eRFID[68].nCardNumber;eRFID[68].bCapCorrectChecked;	eRFID[68].bCapCorrectCheckCameraOK;		eRFID[68].bCapCorrectCheckCameraChecked;		eRFID[68].bCapCorrectCapOn;eRFID[68].bCapCorrectNOK; eRFID[68].bFormPresent; eRFID[68].bBottlePresent; eRFID[68].bDosingTwoPhases; eRFID[68].nDispencerNr; eRFID[68].nDispencerNrSecondPhase; eRFID[68].lrDoseVolumeSV; eRFID[68].lrDoseVolumeCV; eRFID[68].lrDoseVolumeSVSecondPhase; eRFID[68].lrDoseVolumeCVSecondPhase; eRFID[68].bDosed;	eRFID[68].bDoseAborted; eRFID[68].bWeighed; eRFID[68].lrWeightSV; eRFID[68].lrWeightCV; eRFID[68].lrWeightMeasuredCV; eRFID[68].bWeightOK; eRFID[68].bCapPutted; eRFID[68].bCapChecked; eRFID[68].bCapOK; eRFID[68].bCapGripperScrewed; eRFID[68].bCapGripperScrewAborted; eRFID[68].bBottleTransferedToExit; eRFID[68].bBottleTransferedToLabeler; eRFID[68].lrWeightDif; eRFID[68].lrMinWeightCV;eRFID[68].lrMaxWeightCV;
eRFID[69].nCardNumber;eRFID[69].bCapCorrectChecked;	eRFID[69].bCapCorrectCheckCameraOK;		eRFID[69].bCapCorrectCheckCameraChecked;		eRFID[69].bCapCorrectCapOn;eRFID[69].bCapCorrectNOK; eRFID[69].bFormPresent; eRFID[69].bBottlePresent; eRFID[69].bDosingTwoPhases; eRFID[69].nDispencerNr; eRFID[69].nDispencerNrSecondPhase; eRFID[69].lrDoseVolumeSV; eRFID[69].lrDoseVolumeCV; eRFID[69].lrDoseVolumeSVSecondPhase; eRFID[69].lrDoseVolumeCVSecondPhase; eRFID[69].bDosed;	eRFID[69].bDoseAborted; eRFID[69].bWeighed; eRFID[69].lrWeightSV; eRFID[69].lrWeightCV; eRFID[69].lrWeightMeasuredCV; eRFID[69].bWeightOK; eRFID[69].bCapPutted; eRFID[69].bCapChecked; eRFID[69].bCapOK; eRFID[69].bCapGripperScrewed; eRFID[69].bCapGripperScrewAborted; eRFID[69].bBottleTransferedToExit; eRFID[69].bBottleTransferedToLabeler; eRFID[69].lrWeightDif; eRFID[69].lrMinWeightCV;eRFID[69].lrMaxWeightCV;
eRFID[70].nCardNumber;eRFID[70].bCapCorrectChecked;	eRFID[70].bCapCorrectCheckCameraOK;		eRFID[70].bCapCorrectCheckCameraChecked;		eRFID[70].bCapCorrectCapOn;eRFID[70].bCapCorrectNOK; eRFID[70].bFormPresent; eRFID[70].bBottlePresent; eRFID[70].bDosingTwoPhases; eRFID[70].nDispencerNr; eRFID[70].nDispencerNrSecondPhase; eRFID[70].lrDoseVolumeSV; eRFID[70].lrDoseVolumeCV; eRFID[70].lrDoseVolumeSVSecondPhase; eRFID[70].lrDoseVolumeCVSecondPhase; eRFID[70].bDosed;	eRFID[70].bDoseAborted; eRFID[70].bWeighed; eRFID[70].lrWeightSV; eRFID[70].lrWeightCV; eRFID[70].lrWeightMeasuredCV; eRFID[70].bWeightOK; eRFID[70].bCapPutted; eRFID[70].bCapChecked; eRFID[70].bCapOK; eRFID[70].bCapGripperScrewed; eRFID[70].bCapGripperScrewAborted; eRFID[70].bBottleTransferedToExit; eRFID[70].bBottleTransferedToLabeler; eRFID[70].lrWeightDif; eRFID[70].lrMinWeightCV;eRFID[70].lrMaxWeightCV;
eRFID[71].nCardNumber;eRFID[71].bCapCorrectChecked;	eRFID[71].bCapCorrectCheckCameraOK;		eRFID[71].bCapCorrectCheckCameraChecked;		eRFID[71].bCapCorrectCapOn;eRFID[71].bCapCorrectNOK; eRFID[71].bFormPresent; eRFID[71].bBottlePresent; eRFID[71].bDosingTwoPhases; eRFID[71].nDispencerNr; eRFID[71].nDispencerNrSecondPhase; eRFID[71].lrDoseVolumeSV; eRFID[71].lrDoseVolumeCV; eRFID[71].lrDoseVolumeSVSecondPhase; eRFID[71].lrDoseVolumeCVSecondPhase; eRFID[71].bDosed;	eRFID[71].bDoseAborted; eRFID[71].bWeighed; eRFID[71].lrWeightSV; eRFID[71].lrWeightCV; eRFID[71].lrWeightMeasuredCV; eRFID[71].bWeightOK; eRFID[71].bCapPutted; eRFID[71].bCapChecked; eRFID[71].bCapOK; eRFID[71].bCapGripperScrewed; eRFID[71].bCapGripperScrewAborted; eRFID[71].bBottleTransferedToExit; eRFID[71].bBottleTransferedToLabeler; eRFID[71].lrWeightDif; eRFID[71].lrMinWeightCV;eRFID[71].lrMaxWeightCV;
eRFID[72].nCardNumber;eRFID[72].bCapCorrectChecked;	eRFID[72].bCapCorrectCheckCameraOK;		eRFID[72].bCapCorrectCheckCameraChecked;		eRFID[72].bCapCorrectCapOn;eRFID[72].bCapCorrectNOK; eRFID[72].bFormPresent; eRFID[72].bBottlePresent; eRFID[72].bDosingTwoPhases; eRFID[72].nDispencerNr; eRFID[72].nDispencerNrSecondPhase; eRFID[72].lrDoseVolumeSV; eRFID[72].lrDoseVolumeCV; eRFID[72].lrDoseVolumeSVSecondPhase; eRFID[72].lrDoseVolumeCVSecondPhase; eRFID[72].bDosed;	eRFID[72].bDoseAborted; eRFID[72].bWeighed; eRFID[72].lrWeightSV; eRFID[72].lrWeightCV; eRFID[72].lrWeightMeasuredCV; eRFID[72].bWeightOK; eRFID[72].bCapPutted; eRFID[72].bCapChecked; eRFID[72].bCapOK; eRFID[72].bCapGripperScrewed; eRFID[72].bCapGripperScrewAborted; eRFID[72].bBottleTransferedToExit; eRFID[72].bBottleTransferedToLabeler; eRFID[72].lrWeightDif; eRFID[72].lrMinWeightCV;eRFID[72].lrMaxWeightCV;
eRFID[73].nCardNumber;eRFID[73].bCapCorrectChecked;	eRFID[73].bCapCorrectCheckCameraOK;		eRFID[73].bCapCorrectCheckCameraChecked;		eRFID[73].bCapCorrectCapOn;eRFID[73].bCapCorrectNOK; eRFID[73].bFormPresent; eRFID[73].bBottlePresent; eRFID[73].bDosingTwoPhases; eRFID[73].nDispencerNr; eRFID[73].nDispencerNrSecondPhase; eRFID[73].lrDoseVolumeSV; eRFID[73].lrDoseVolumeCV; eRFID[73].lrDoseVolumeSVSecondPhase; eRFID[73].lrDoseVolumeCVSecondPhase; eRFID[73].bDosed;	eRFID[73].bDoseAborted; eRFID[73].bWeighed; eRFID[73].lrWeightSV; eRFID[73].lrWeightCV; eRFID[73].lrWeightMeasuredCV; eRFID[73].bWeightOK; eRFID[73].bCapPutted; eRFID[73].bCapChecked; eRFID[73].bCapOK; eRFID[73].bCapGripperScrewed; eRFID[73].bCapGripperScrewAborted; eRFID[73].bBottleTransferedToExit; eRFID[73].bBottleTransferedToLabeler; eRFID[73].lrWeightDif; eRFID[73].lrMinWeightCV;eRFID[73].lrMaxWeightCV;
eRFID[74].nCardNumber;eRFID[74].bCapCorrectChecked;	eRFID[74].bCapCorrectCheckCameraOK;		eRFID[74].bCapCorrectCheckCameraChecked;		eRFID[74].bCapCorrectCapOn;eRFID[74].bCapCorrectNOK; eRFID[74].bFormPresent; eRFID[74].bBottlePresent; eRFID[74].bDosingTwoPhases; eRFID[74].nDispencerNr; eRFID[74].nDispencerNrSecondPhase; eRFID[74].lrDoseVolumeSV; eRFID[74].lrDoseVolumeCV; eRFID[74].lrDoseVolumeSVSecondPhase; eRFID[74].lrDoseVolumeCVSecondPhase; eRFID[74].bDosed;	eRFID[74].bDoseAborted; eRFID[74].bWeighed; eRFID[74].lrWeightSV; eRFID[74].lrWeightCV; eRFID[74].lrWeightMeasuredCV; eRFID[74].bWeightOK; eRFID[74].bCapPutted; eRFID[74].bCapChecked; eRFID[74].bCapOK; eRFID[74].bCapGripperScrewed; eRFID[74].bCapGripperScrewAborted; eRFID[74].bBottleTransferedToExit; eRFID[74].bBottleTransferedToLabeler; eRFID[74].lrWeightDif; eRFID[74].lrMinWeightCV;eRFID[74].lrMaxWeightCV;
eRFID[75].nCardNumber;eRFID[75].bCapCorrectChecked;	eRFID[75].bCapCorrectCheckCameraOK;		eRFID[75].bCapCorrectCheckCameraChecked;		eRFID[75].bCapCorrectCapOn;eRFID[75].bCapCorrectNOK; eRFID[75].bFormPresent; eRFID[75].bBottlePresent; eRFID[75].bDosingTwoPhases; eRFID[75].nDispencerNr; eRFID[75].nDispencerNrSecondPhase; eRFID[75].lrDoseVolumeSV; eRFID[75].lrDoseVolumeCV; eRFID[75].lrDoseVolumeSVSecondPhase; eRFID[75].lrDoseVolumeCVSecondPhase; eRFID[75].bDosed;	eRFID[75].bDoseAborted; eRFID[75].bWeighed; eRFID[75].lrWeightSV; eRFID[75].lrWeightCV; eRFID[75].lrWeightMeasuredCV; eRFID[75].bWeightOK; eRFID[75].bCapPutted; eRFID[75].bCapChecked; eRFID[75].bCapOK; eRFID[75].bCapGripperScrewed; eRFID[75].bCapGripperScrewAborted; eRFID[75].bBottleTransferedToExit; eRFID[75].bBottleTransferedToLabeler; eRFID[75].lrWeightDif; eRFID[75].lrMinWeightCV;eRFID[75].lrMaxWeightCV;
eRFID[76].nCardNumber;eRFID[76].bCapCorrectChecked;	eRFID[76].bCapCorrectCheckCameraOK;		eRFID[76].bCapCorrectCheckCameraChecked;		eRFID[76].bCapCorrectCapOn;eRFID[76].bCapCorrectNOK; eRFID[76].bFormPresent; eRFID[76].bBottlePresent; eRFID[76].bDosingTwoPhases; eRFID[76].nDispencerNr; eRFID[76].nDispencerNrSecondPhase; eRFID[76].lrDoseVolumeSV; eRFID[76].lrDoseVolumeCV; eRFID[76].lrDoseVolumeSVSecondPhase; eRFID[76].lrDoseVolumeCVSecondPhase; eRFID[76].bDosed;	eRFID[76].bDoseAborted; eRFID[76].bWeighed; eRFID[76].lrWeightSV; eRFID[76].lrWeightCV; eRFID[76].lrWeightMeasuredCV; eRFID[76].bWeightOK; eRFID[76].bCapPutted; eRFID[76].bCapChecked; eRFID[76].bCapOK; eRFID[76].bCapGripperScrewed; eRFID[76].bCapGripperScrewAborted; eRFID[76].bBottleTransferedToExit; eRFID[76].bBottleTransferedToLabeler; eRFID[76].lrWeightDif; eRFID[76].lrMinWeightCV;eRFID[76].lrMaxWeightCV;
eRFID[77].nCardNumber;eRFID[77].bCapCorrectChecked;	eRFID[77].bCapCorrectCheckCameraOK;		eRFID[77].bCapCorrectCheckCameraChecked;		eRFID[77].bCapCorrectCapOn;eRFID[77].bCapCorrectNOK; eRFID[77].bFormPresent; eRFID[77].bBottlePresent; eRFID[77].bDosingTwoPhases; eRFID[77].nDispencerNr; eRFID[77].nDispencerNrSecondPhase; eRFID[77].lrDoseVolumeSV; eRFID[77].lrDoseVolumeCV; eRFID[77].lrDoseVolumeSVSecondPhase; eRFID[77].lrDoseVolumeCVSecondPhase; eRFID[77].bDosed;	eRFID[77].bDoseAborted; eRFID[77].bWeighed; eRFID[77].lrWeightSV; eRFID[77].lrWeightCV; eRFID[77].lrWeightMeasuredCV; eRFID[77].bWeightOK; eRFID[77].bCapPutted; eRFID[77].bCapChecked; eRFID[77].bCapOK; eRFID[77].bCapGripperScrewed; eRFID[77].bCapGripperScrewAborted; eRFID[77].bBottleTransferedToExit; eRFID[77].bBottleTransferedToLabeler; eRFID[77].lrWeightDif; eRFID[77].lrMinWeightCV;eRFID[77].lrMaxWeightCV;
eRFID[78].nCardNumber;eRFID[78].bCapCorrectChecked;	eRFID[78].bCapCorrectCheckCameraOK;		eRFID[78].bCapCorrectCheckCameraChecked;		eRFID[78].bCapCorrectCapOn;eRFID[78].bCapCorrectNOK; eRFID[78].bFormPresent; eRFID[78].bBottlePresent; eRFID[78].bDosingTwoPhases; eRFID[78].nDispencerNr; eRFID[78].nDispencerNrSecondPhase; eRFID[78].lrDoseVolumeSV; eRFID[78].lrDoseVolumeCV; eRFID[78].lrDoseVolumeSVSecondPhase; eRFID[78].lrDoseVolumeCVSecondPhase; eRFID[78].bDosed;	eRFID[78].bDoseAborted; eRFID[78].bWeighed; eRFID[78].lrWeightSV; eRFID[78].lrWeightCV; eRFID[78].lrWeightMeasuredCV; eRFID[78].bWeightOK; eRFID[78].bCapPutted; eRFID[78].bCapChecked; eRFID[78].bCapOK; eRFID[78].bCapGripperScrewed; eRFID[78].bCapGripperScrewAborted; eRFID[78].bBottleTransferedToExit; eRFID[78].bBottleTransferedToLabeler; eRFID[78].lrWeightDif; eRFID[78].lrMinWeightCV;eRFID[78].lrMaxWeightCV;
eRFID[79].nCardNumber;eRFID[79].bCapCorrectChecked;	eRFID[79].bCapCorrectCheckCameraOK;		eRFID[79].bCapCorrectCheckCameraChecked;		eRFID[79].bCapCorrectCapOn;eRFID[79].bCapCorrectNOK; eRFID[79].bFormPresent; eRFID[79].bBottlePresent; eRFID[79].bDosingTwoPhases; eRFID[79].nDispencerNr; eRFID[79].nDispencerNrSecondPhase; eRFID[79].lrDoseVolumeSV; eRFID[79].lrDoseVolumeCV; eRFID[79].lrDoseVolumeSVSecondPhase; eRFID[79].lrDoseVolumeCVSecondPhase; eRFID[79].bDosed;	eRFID[79].bDoseAborted; eRFID[79].bWeighed; eRFID[79].lrWeightSV; eRFID[79].lrWeightCV; eRFID[79].lrWeightMeasuredCV; eRFID[79].bWeightOK; eRFID[79].bCapPutted; eRFID[79].bCapChecked; eRFID[79].bCapOK; eRFID[79].bCapGripperScrewed; eRFID[79].bCapGripperScrewAborted; eRFID[79].bBottleTransferedToExit; eRFID[79].bBottleTransferedToLabeler; eRFID[79].lrWeightDif; eRFID[79].lrMinWeightCV;eRFID[79].lrMaxWeightCV;
eRFID[80].nCardNumber;eRFID[80].bCapCorrectChecked;	eRFID[80].bCapCorrectCheckCameraOK;		eRFID[80].bCapCorrectCheckCameraChecked;		eRFID[80].bCapCorrectCapOn;eRFID[80].bCapCorrectNOK; eRFID[80].bFormPresent; eRFID[80].bBottlePresent; eRFID[80].bDosingTwoPhases; eRFID[80].nDispencerNr; eRFID[80].nDispencerNrSecondPhase; eRFID[80].lrDoseVolumeSV; eRFID[80].lrDoseVolumeCV; eRFID[80].lrDoseVolumeSVSecondPhase; eRFID[80].lrDoseVolumeCVSecondPhase; eRFID[80].bDosed;	eRFID[80].bDoseAborted; eRFID[80].bWeighed; eRFID[80].lrWeightSV; eRFID[80].lrWeightCV; eRFID[80].lrWeightMeasuredCV; eRFID[80].bWeightOK; eRFID[80].bCapPutted; eRFID[80].bCapChecked; eRFID[80].bCapOK; eRFID[80].bCapGripperScrewed; eRFID[80].bCapGripperScrewAborted; eRFID[80].bBottleTransferedToExit; eRFID[80].bBottleTransferedToLabeler; eRFID[80].lrWeightDif; eRFID[80].lrMinWeightCV;eRFID[80].lrMaxWeightCV;
eRFID[81].nCardNumber;eRFID[81].bCapCorrectChecked;	eRFID[81].bCapCorrectCheckCameraOK;		eRFID[81].bCapCorrectCheckCameraChecked;		eRFID[81].bCapCorrectCapOn;eRFID[81].bCapCorrectNOK; eRFID[81].bFormPresent; eRFID[81].bBottlePresent; eRFID[81].bDosingTwoPhases; eRFID[81].nDispencerNr; eRFID[81].nDispencerNrSecondPhase; eRFID[81].lrDoseVolumeSV; eRFID[81].lrDoseVolumeCV; eRFID[81].lrDoseVolumeSVSecondPhase; eRFID[81].lrDoseVolumeCVSecondPhase; eRFID[81].bDosed;	eRFID[81].bDoseAborted; eRFID[81].bWeighed; eRFID[81].lrWeightSV; eRFID[81].lrWeightCV; eRFID[81].lrWeightMeasuredCV; eRFID[81].bWeightOK; eRFID[81].bCapPutted; eRFID[81].bCapChecked; eRFID[81].bCapOK; eRFID[81].bCapGripperScrewed; eRFID[81].bCapGripperScrewAborted; eRFID[81].bBottleTransferedToExit; eRFID[81].bBottleTransferedToLabeler; eRFID[81].lrWeightDif; eRFID[81].lrMinWeightCV;eRFID[81].lrMaxWeightCV;
eRFID[82].nCardNumber;eRFID[82].bCapCorrectChecked;	eRFID[82].bCapCorrectCheckCameraOK;		eRFID[82].bCapCorrectCheckCameraChecked;		eRFID[82].bCapCorrectCapOn;eRFID[82].bCapCorrectNOK; eRFID[82].bFormPresent; eRFID[82].bBottlePresent; eRFID[82].bDosingTwoPhases; eRFID[82].nDispencerNr; eRFID[82].nDispencerNrSecondPhase; eRFID[82].lrDoseVolumeSV; eRFID[82].lrDoseVolumeCV; eRFID[82].lrDoseVolumeSVSecondPhase; eRFID[82].lrDoseVolumeCVSecondPhase; eRFID[82].bDosed;	eRFID[82].bDoseAborted; eRFID[82].bWeighed; eRFID[82].lrWeightSV; eRFID[82].lrWeightCV; eRFID[82].lrWeightMeasuredCV; eRFID[82].bWeightOK; eRFID[82].bCapPutted; eRFID[82].bCapChecked; eRFID[82].bCapOK; eRFID[82].bCapGripperScrewed; eRFID[82].bCapGripperScrewAborted; eRFID[82].bBottleTransferedToExit; eRFID[82].bBottleTransferedToLabeler; eRFID[82].lrWeightDif; eRFID[82].lrMinWeightCV;eRFID[82].lrMaxWeightCV;
eRFID[83].nCardNumber;eRFID[83].bCapCorrectChecked;	eRFID[83].bCapCorrectCheckCameraOK;		eRFID[83].bCapCorrectCheckCameraChecked;		eRFID[83].bCapCorrectCapOn;eRFID[83].bCapCorrectNOK; eRFID[83].bFormPresent; eRFID[83].bBottlePresent; eRFID[83].bDosingTwoPhases; eRFID[83].nDispencerNr; eRFID[83].nDispencerNrSecondPhase; eRFID[83].lrDoseVolumeSV; eRFID[83].lrDoseVolumeCV; eRFID[83].lrDoseVolumeSVSecondPhase; eRFID[83].lrDoseVolumeCVSecondPhase; eRFID[83].bDosed;	eRFID[83].bDoseAborted; eRFID[83].bWeighed; eRFID[83].lrWeightSV; eRFID[83].lrWeightCV; eRFID[83].lrWeightMeasuredCV; eRFID[83].bWeightOK; eRFID[83].bCapPutted; eRFID[83].bCapChecked; eRFID[83].bCapOK; eRFID[83].bCapGripperScrewed; eRFID[83].bCapGripperScrewAborted; eRFID[83].bBottleTransferedToExit; eRFID[83].bBottleTransferedToLabeler; eRFID[83].lrWeightDif; eRFID[83].lrMinWeightCV;eRFID[83].lrMaxWeightCV;
eRFID[84].nCardNumber;eRFID[84].bCapCorrectChecked;	eRFID[84].bCapCorrectCheckCameraOK;		eRFID[84].bCapCorrectCheckCameraChecked;		eRFID[84].bCapCorrectCapOn;eRFID[84].bCapCorrectNOK; eRFID[84].bFormPresent; eRFID[84].bBottlePresent; eRFID[84].bDosingTwoPhases; eRFID[84].nDispencerNr; eRFID[84].nDispencerNrSecondPhase; eRFID[84].lrDoseVolumeSV; eRFID[84].lrDoseVolumeCV; eRFID[84].lrDoseVolumeSVSecondPhase; eRFID[84].lrDoseVolumeCVSecondPhase; eRFID[84].bDosed;	eRFID[84].bDoseAborted; eRFID[84].bWeighed; eRFID[84].lrWeightSV; eRFID[84].lrWeightCV; eRFID[84].lrWeightMeasuredCV; eRFID[84].bWeightOK; eRFID[84].bCapPutted; eRFID[84].bCapChecked; eRFID[84].bCapOK; eRFID[84].bCapGripperScrewed; eRFID[84].bCapGripperScrewAborted; eRFID[84].bBottleTransferedToExit; eRFID[84].bBottleTransferedToLabeler; eRFID[84].lrWeightDif; eRFID[84].lrMinWeightCV;eRFID[84].lrMaxWeightCV;
eRFID[85].nCardNumber;eRFID[85].bCapCorrectChecked;	eRFID[85].bCapCorrectCheckCameraOK;		eRFID[85].bCapCorrectCheckCameraChecked;		eRFID[85].bCapCorrectCapOn;eRFID[85].bCapCorrectNOK; eRFID[85].bFormPresent; eRFID[85].bBottlePresent; eRFID[85].bDosingTwoPhases; eRFID[85].nDispencerNr; eRFID[85].nDispencerNrSecondPhase; eRFID[85].lrDoseVolumeSV; eRFID[85].lrDoseVolumeCV; eRFID[85].lrDoseVolumeSVSecondPhase; eRFID[85].lrDoseVolumeCVSecondPhase; eRFID[85].bDosed;	eRFID[85].bDoseAborted; eRFID[85].bWeighed; eRFID[85].lrWeightSV; eRFID[85].lrWeightCV; eRFID[85].lrWeightMeasuredCV; eRFID[85].bWeightOK; eRFID[85].bCapPutted; eRFID[85].bCapChecked; eRFID[85].bCapOK; eRFID[85].bCapGripperScrewed; eRFID[85].bCapGripperScrewAborted; eRFID[85].bBottleTransferedToExit; eRFID[85].bBottleTransferedToLabeler; eRFID[85].lrWeightDif; eRFID[85].lrMinWeightCV;eRFID[85].lrMaxWeightCV;
eRFID[86].nCardNumber;eRFID[86].bCapCorrectChecked;	eRFID[86].bCapCorrectCheckCameraOK;		eRFID[86].bCapCorrectCheckCameraChecked;		eRFID[86].bCapCorrectCapOn;eRFID[86].bCapCorrectNOK; eRFID[86].bFormPresent; eRFID[86].bBottlePresent; eRFID[86].bDosingTwoPhases; eRFID[86].nDispencerNr; eRFID[86].nDispencerNrSecondPhase; eRFID[86].lrDoseVolumeSV; eRFID[86].lrDoseVolumeCV; eRFID[86].lrDoseVolumeSVSecondPhase; eRFID[86].lrDoseVolumeCVSecondPhase; eRFID[86].bDosed;	eRFID[86].bDoseAborted; eRFID[86].bWeighed; eRFID[86].lrWeightSV; eRFID[86].lrWeightCV; eRFID[86].lrWeightMeasuredCV; eRFID[86].bWeightOK; eRFID[86].bCapPutted; eRFID[86].bCapChecked; eRFID[86].bCapOK; eRFID[86].bCapGripperScrewed; eRFID[86].bCapGripperScrewAborted; eRFID[86].bBottleTransferedToExit; eRFID[86].bBottleTransferedToLabeler; eRFID[86].lrWeightDif; eRFID[86].lrMinWeightCV;eRFID[86].lrMaxWeightCV;
eRFID[87].nCardNumber;eRFID[87].bCapCorrectChecked;	eRFID[87].bCapCorrectCheckCameraOK;		eRFID[87].bCapCorrectCheckCameraChecked;		eRFID[87].bCapCorrectCapOn;eRFID[87].bCapCorrectNOK; eRFID[87].bFormPresent; eRFID[87].bBottlePresent; eRFID[87].bDosingTwoPhases; eRFID[87].nDispencerNr; eRFID[87].nDispencerNrSecondPhase; eRFID[87].lrDoseVolumeSV; eRFID[87].lrDoseVolumeCV; eRFID[87].lrDoseVolumeSVSecondPhase; eRFID[87].lrDoseVolumeCVSecondPhase; eRFID[87].bDosed;	eRFID[87].bDoseAborted; eRFID[87].bWeighed; eRFID[87].lrWeightSV; eRFID[87].lrWeightCV; eRFID[87].lrWeightMeasuredCV; eRFID[87].bWeightOK; eRFID[87].bCapPutted; eRFID[87].bCapChecked; eRFID[87].bCapOK; eRFID[87].bCapGripperScrewed; eRFID[87].bCapGripperScrewAborted; eRFID[87].bBottleTransferedToExit; eRFID[87].bBottleTransferedToLabeler; eRFID[87].lrWeightDif; eRFID[87].lrMinWeightCV;eRFID[87].lrMaxWeightCV;
eRFID[88].nCardNumber;eRFID[88].bCapCorrectChecked;	eRFID[88].bCapCorrectCheckCameraOK;		eRFID[88].bCapCorrectCheckCameraChecked;		eRFID[88].bCapCorrectCapOn;eRFID[88].bCapCorrectNOK; eRFID[88].bFormPresent; eRFID[88].bBottlePresent; eRFID[88].bDosingTwoPhases; eRFID[88].nDispencerNr; eRFID[88].nDispencerNrSecondPhase; eRFID[88].lrDoseVolumeSV; eRFID[88].lrDoseVolumeCV; eRFID[88].lrDoseVolumeSVSecondPhase; eRFID[88].lrDoseVolumeCVSecondPhase; eRFID[88].bDosed;	eRFID[88].bDoseAborted; eRFID[88].bWeighed; eRFID[88].lrWeightSV; eRFID[88].lrWeightCV; eRFID[88].lrWeightMeasuredCV; eRFID[88].bWeightOK; eRFID[88].bCapPutted; eRFID[88].bCapChecked; eRFID[88].bCapOK; eRFID[88].bCapGripperScrewed; eRFID[88].bCapGripperScrewAborted; eRFID[88].bBottleTransferedToExit; eRFID[88].bBottleTransferedToLabeler; eRFID[88].lrWeightDif; eRFID[88].lrMinWeightCV;eRFID[88].lrMaxWeightCV;
eRFID[89].nCardNumber;eRFID[89].bCapCorrectChecked;	eRFID[89].bCapCorrectCheckCameraOK;		eRFID[89].bCapCorrectCheckCameraChecked;		eRFID[89].bCapCorrectCapOn;eRFID[89].bCapCorrectNOK; eRFID[89].bFormPresent; eRFID[89].bBottlePresent; eRFID[89].bDosingTwoPhases; eRFID[89].nDispencerNr; eRFID[89].nDispencerNrSecondPhase; eRFID[89].lrDoseVolumeSV; eRFID[89].lrDoseVolumeCV; eRFID[89].lrDoseVolumeSVSecondPhase; eRFID[89].lrDoseVolumeCVSecondPhase; eRFID[89].bDosed;	eRFID[89].bDoseAborted; eRFID[89].bWeighed; eRFID[89].lrWeightSV; eRFID[89].lrWeightCV; eRFID[89].lrWeightMeasuredCV; eRFID[89].bWeightOK; eRFID[89].bCapPutted; eRFID[89].bCapChecked; eRFID[89].bCapOK; eRFID[89].bCapGripperScrewed; eRFID[89].bCapGripperScrewAborted; eRFID[89].bBottleTransferedToExit; eRFID[89].bBottleTransferedToLabeler; eRFID[89].lrWeightDif; eRFID[89].lrMinWeightCV;eRFID[89].lrMaxWeightCV;
eRFID[90].nCardNumber;eRFID[90].bCapCorrectChecked;	eRFID[90].bCapCorrectCheckCameraOK;		eRFID[90].bCapCorrectCheckCameraChecked;		eRFID[90].bCapCorrectCapOn;eRFID[90].bCapCorrectNOK; eRFID[90].bFormPresent; eRFID[90].bBottlePresent; eRFID[90].bDosingTwoPhases; eRFID[90].nDispencerNr; eRFID[90].nDispencerNrSecondPhase; eRFID[90].lrDoseVolumeSV; eRFID[90].lrDoseVolumeCV; eRFID[90].lrDoseVolumeSVSecondPhase; eRFID[90].lrDoseVolumeCVSecondPhase; eRFID[90].bDosed;	eRFID[90].bDoseAborted; eRFID[90].bWeighed; eRFID[90].lrWeightSV; eRFID[90].lrWeightCV; eRFID[90].lrWeightMeasuredCV; eRFID[90].bWeightOK; eRFID[90].bCapPutted; eRFID[90].bCapChecked; eRFID[90].bCapOK; eRFID[90].bCapGripperScrewed; eRFID[90].bCapGripperScrewAborted; eRFID[90].bBottleTransferedToExit; eRFID[90].bBottleTransferedToLabeler; eRFID[90].lrWeightDif; eRFID[90].lrMinWeightCV;eRFID[90].lrMaxWeightCV;
eRFID[91].nCardNumber;eRFID[91].bCapCorrectChecked;	eRFID[91].bCapCorrectCheckCameraOK;		eRFID[91].bCapCorrectCheckCameraChecked;		eRFID[91].bCapCorrectCapOn;eRFID[91].bCapCorrectNOK; eRFID[91].bFormPresent; eRFID[91].bBottlePresent; eRFID[91].bDosingTwoPhases; eRFID[91].nDispencerNr; eRFID[91].nDispencerNrSecondPhase; eRFID[91].lrDoseVolumeSV; eRFID[91].lrDoseVolumeCV; eRFID[91].lrDoseVolumeSVSecondPhase; eRFID[91].lrDoseVolumeCVSecondPhase; eRFID[91].bDosed;	eRFID[91].bDoseAborted; eRFID[91].bWeighed; eRFID[91].lrWeightSV; eRFID[91].lrWeightCV; eRFID[91].lrWeightMeasuredCV; eRFID[91].bWeightOK; eRFID[91].bCapPutted; eRFID[91].bCapChecked; eRFID[91].bCapOK; eRFID[91].bCapGripperScrewed; eRFID[91].bCapGripperScrewAborted; eRFID[91].bBottleTransferedToExit; eRFID[91].bBottleTransferedToLabeler; eRFID[91].lrWeightDif; eRFID[91].lrMinWeightCV;eRFID[91].lrMaxWeightCV;
eRFID[92].nCardNumber;eRFID[92].bCapCorrectChecked;	eRFID[92].bCapCorrectCheckCameraOK;		eRFID[92].bCapCorrectCheckCameraChecked;		eRFID[92].bCapCorrectCapOn;eRFID[92].bCapCorrectNOK; eRFID[92].bFormPresent; eRFID[92].bBottlePresent; eRFID[92].bDosingTwoPhases; eRFID[92].nDispencerNr; eRFID[92].nDispencerNrSecondPhase; eRFID[92].lrDoseVolumeSV; eRFID[92].lrDoseVolumeCV; eRFID[92].lrDoseVolumeSVSecondPhase; eRFID[92].lrDoseVolumeCVSecondPhase; eRFID[92].bDosed;	eRFID[92].bDoseAborted; eRFID[92].bWeighed; eRFID[92].lrWeightSV; eRFID[92].lrWeightCV; eRFID[92].lrWeightMeasuredCV; eRFID[92].bWeightOK; eRFID[92].bCapPutted; eRFID[92].bCapChecked; eRFID[92].bCapOK; eRFID[92].bCapGripperScrewed; eRFID[92].bCapGripperScrewAborted; eRFID[92].bBottleTransferedToExit; eRFID[92].bBottleTransferedToLabeler; eRFID[92].lrWeightDif; eRFID[92].lrMinWeightCV;eRFID[92].lrMaxWeightCV;
eRFID[93].nCardNumber;eRFID[93].bCapCorrectChecked;	eRFID[93].bCapCorrectCheckCameraOK;		eRFID[93].bCapCorrectCheckCameraChecked;		eRFID[93].bCapCorrectCapOn;eRFID[93].bCapCorrectNOK; eRFID[93].bFormPresent; eRFID[93].bBottlePresent; eRFID[93].bDosingTwoPhases; eRFID[93].nDispencerNr; eRFID[93].nDispencerNrSecondPhase; eRFID[93].lrDoseVolumeSV; eRFID[93].lrDoseVolumeCV; eRFID[93].lrDoseVolumeSVSecondPhase; eRFID[93].lrDoseVolumeCVSecondPhase; eRFID[93].bDosed;	eRFID[93].bDoseAborted; eRFID[93].bWeighed; eRFID[93].lrWeightSV; eRFID[93].lrWeightCV; eRFID[93].lrWeightMeasuredCV; eRFID[93].bWeightOK; eRFID[93].bCapPutted; eRFID[93].bCapChecked; eRFID[93].bCapOK; eRFID[93].bCapGripperScrewed; eRFID[93].bCapGripperScrewAborted; eRFID[93].bBottleTransferedToExit; eRFID[93].bBottleTransferedToLabeler; eRFID[93].lrWeightDif; eRFID[93].lrMinWeightCV;eRFID[93].lrMaxWeightCV;
eRFID[94].nCardNumber;eRFID[94].bCapCorrectChecked;	eRFID[94].bCapCorrectCheckCameraOK;		eRFID[94].bCapCorrectCheckCameraChecked;		eRFID[94].bCapCorrectCapOn;eRFID[94].bCapCorrectNOK; eRFID[94].bFormPresent; eRFID[94].bBottlePresent; eRFID[94].bDosingTwoPhases; eRFID[94].nDispencerNr; eRFID[94].nDispencerNrSecondPhase; eRFID[94].lrDoseVolumeSV; eRFID[94].lrDoseVolumeCV; eRFID[94].lrDoseVolumeSVSecondPhase; eRFID[94].lrDoseVolumeCVSecondPhase; eRFID[94].bDosed;	eRFID[94].bDoseAborted; eRFID[94].bWeighed; eRFID[94].lrWeightSV; eRFID[94].lrWeightCV; eRFID[94].lrWeightMeasuredCV; eRFID[94].bWeightOK; eRFID[94].bCapPutted; eRFID[94].bCapChecked; eRFID[94].bCapOK; eRFID[94].bCapGripperScrewed; eRFID[94].bCapGripperScrewAborted; eRFID[94].bBottleTransferedToExit; eRFID[94].bBottleTransferedToLabeler; eRFID[94].lrWeightDif; eRFID[94].lrMinWeightCV;eRFID[94].lrMaxWeightCV;
eRFID[95].nCardNumber;eRFID[95].bCapCorrectChecked;	eRFID[95].bCapCorrectCheckCameraOK;		eRFID[95].bCapCorrectCheckCameraChecked;		eRFID[95].bCapCorrectCapOn;eRFID[95].bCapCorrectNOK; eRFID[95].bFormPresent; eRFID[95].bBottlePresent; eRFID[95].bDosingTwoPhases; eRFID[95].nDispencerNr; eRFID[95].nDispencerNrSecondPhase; eRFID[95].lrDoseVolumeSV; eRFID[95].lrDoseVolumeCV; eRFID[95].lrDoseVolumeSVSecondPhase; eRFID[95].lrDoseVolumeCVSecondPhase; eRFID[95].bDosed;	eRFID[95].bDoseAborted; eRFID[95].bWeighed; eRFID[95].lrWeightSV; eRFID[95].lrWeightCV; eRFID[95].lrWeightMeasuredCV; eRFID[95].bWeightOK; eRFID[95].bCapPutted; eRFID[95].bCapChecked; eRFID[95].bCapOK; eRFID[95].bCapGripperScrewed; eRFID[95].bCapGripperScrewAborted; eRFID[95].bBottleTransferedToExit; eRFID[95].bBottleTransferedToLabeler; eRFID[95].lrWeightDif; eRFID[95].lrMinWeightCV;eRFID[95].lrMaxWeightCV;
eRFID[96].nCardNumber;eRFID[96].bCapCorrectChecked;	eRFID[96].bCapCorrectCheckCameraOK;		eRFID[96].bCapCorrectCheckCameraChecked;		eRFID[96].bCapCorrectCapOn;eRFID[96].bCapCorrectNOK; eRFID[96].bFormPresent; eRFID[96].bBottlePresent; eRFID[96].bDosingTwoPhases; eRFID[96].nDispencerNr; eRFID[96].nDispencerNrSecondPhase; eRFID[96].lrDoseVolumeSV; eRFID[96].lrDoseVolumeCV; eRFID[96].lrDoseVolumeSVSecondPhase; eRFID[96].lrDoseVolumeCVSecondPhase; eRFID[96].bDosed;	eRFID[96].bDoseAborted; eRFID[96].bWeighed; eRFID[96].lrWeightSV; eRFID[96].lrWeightCV; eRFID[96].lrWeightMeasuredCV; eRFID[96].bWeightOK; eRFID[96].bCapPutted; eRFID[96].bCapChecked; eRFID[96].bCapOK; eRFID[96].bCapGripperScrewed; eRFID[96].bCapGripperScrewAborted; eRFID[96].bBottleTransferedToExit; eRFID[96].bBottleTransferedToLabeler; eRFID[96].lrWeightDif; eRFID[96].lrMinWeightCV;eRFID[96].lrMaxWeightCV;
eRFID[97].nCardNumber;eRFID[97].bCapCorrectChecked;	eRFID[97].bCapCorrectCheckCameraOK;		eRFID[97].bCapCorrectCheckCameraChecked;		eRFID[97].bCapCorrectCapOn;eRFID[97].bCapCorrectNOK; eRFID[97].bFormPresent; eRFID[97].bBottlePresent; eRFID[97].bDosingTwoPhases; eRFID[97].nDispencerNr; eRFID[97].nDispencerNrSecondPhase; eRFID[97].lrDoseVolumeSV; eRFID[97].lrDoseVolumeCV; eRFID[97].lrDoseVolumeSVSecondPhase; eRFID[97].lrDoseVolumeCVSecondPhase; eRFID[97].bDosed;	eRFID[97].bDoseAborted; eRFID[97].bWeighed; eRFID[97].lrWeightSV; eRFID[97].lrWeightCV; eRFID[97].lrWeightMeasuredCV; eRFID[97].bWeightOK; eRFID[97].bCapPutted; eRFID[97].bCapChecked; eRFID[97].bCapOK; eRFID[97].bCapGripperScrewed; eRFID[97].bCapGripperScrewAborted; eRFID[97].bBottleTransferedToExit; eRFID[97].bBottleTransferedToLabeler; eRFID[97].lrWeightDif; eRFID[97].lrMinWeightCV;eRFID[97].lrMaxWeightCV;
eRFID[98].nCardNumber;eRFID[98].bCapCorrectChecked;	eRFID[98].bCapCorrectCheckCameraOK;		eRFID[98].bCapCorrectCheckCameraChecked;		eRFID[98].bCapCorrectCapOn;eRFID[98].bCapCorrectNOK; eRFID[98].bFormPresent; eRFID[98].bBottlePresent; eRFID[98].bDosingTwoPhases; eRFID[98].nDispencerNr; eRFID[98].nDispencerNrSecondPhase; eRFID[98].lrDoseVolumeSV; eRFID[98].lrDoseVolumeCV; eRFID[98].lrDoseVolumeSVSecondPhase; eRFID[98].lrDoseVolumeCVSecondPhase; eRFID[98].bDosed;	eRFID[98].bDoseAborted; eRFID[98].bWeighed; eRFID[98].lrWeightSV; eRFID[98].lrWeightCV; eRFID[98].lrWeightMeasuredCV; eRFID[98].bWeightOK; eRFID[98].bCapPutted; eRFID[98].bCapChecked; eRFID[98].bCapOK; eRFID[98].bCapGripperScrewed; eRFID[98].bCapGripperScrewAborted; eRFID[98].bBottleTransferedToExit; eRFID[98].bBottleTransferedToLabeler; eRFID[98].lrWeightDif; eRFID[98].lrMinWeightCV;eRFID[98].lrMaxWeightCV;
eRFID[99].nCardNumber;eRFID[99].bCapCorrectChecked;	eRFID[99].bCapCorrectCheckCameraOK;		eRFID[99].bCapCorrectCheckCameraChecked;		eRFID[99].bCapCorrectCapOn;eRFID[99].bCapCorrectNOK; eRFID[99].bFormPresent; eRFID[99].bBottlePresent; eRFID[99].bDosingTwoPhases; eRFID[99].nDispencerNr; eRFID[99].nDispencerNrSecondPhase; eRFID[99].lrDoseVolumeSV; eRFID[99].lrDoseVolumeCV; eRFID[99].lrDoseVolumeSVSecondPhase; eRFID[99].lrDoseVolumeCVSecondPhase; eRFID[99].bDosed;	eRFID[99].bDoseAborted; eRFID[99].bWeighed; eRFID[99].lrWeightSV; eRFID[99].lrWeightCV; eRFID[99].lrWeightMeasuredCV; eRFID[99].bWeightOK; eRFID[99].bCapPutted; eRFID[99].bCapChecked; eRFID[99].bCapOK; eRFID[99].bCapGripperScrewed; eRFID[99].bCapGripperScrewAborted; eRFID[99].bBottleTransferedToExit; eRFID[99].bBottleTransferedToLabeler; eRFID[99].lrWeightDif; eRFID[99].lrMinWeightCV;eRFID[99].lrMaxWeightCV;
eRFID[100].nCardNumber;eRFID[100].bCapCorrectChecked;eRFID[100].bCapCorrectCheckCameraOK;;	eRFID[100].bCapCorrectCheckCameraChecked;;		eRFID[100].bCapCorrectCapOn;eRFID[100].bCapCorrectNOK;eRFID[100].bFormPresent; eRFID[100].bBottlePresent; eRFID[100].bDosingTwoPhases; eRFID[100].nDispencerNr; eRFID[100].nDispencerNrSecondPhase; eRFID[100].lrDoseVolumeSV; eRFID[100].lrDoseVolumeCV; eRFID[100].lrDoseVolumeSVSecondPhase; eRFID[100].lrDoseVolumeCVSecondPhase; eRFID[100].bDoseAborted; eRFID[100].bWeighed; eRFID[100].lrWeightSV; eRFID[100].lrWeightCV; eRFID[100].lrWeightMeasuredCV; eRFID[100].bWeightOK; eRFID[100].bCapPutted; eRFID[100].bCapChecked; eRFID[100].bCapOK; eRFID[100].bCapGripperScrewed; eRFID[100].bCapGripperScrewAborted; eRFID[100].bBottleTransferedToExit; eRFID[100].bBottleTransferedToLabeler; eRFID[100].lrWeightDif; eRFID[100].lrMinWeightCV;eRFID[100].lrMinWeightCV;;


IF GVL.bV1Hz THEN
	FOR i := 1 TO 100 DO
		IF eRFID[i].nCardNumber = 544 THEN
			iPodglad := i;
		END_IF
	END_FOR
END_IF
IF iPodglad = 0 THEN
	 iPodglad := 100;
END_IF
;eRFID[iPodglad].nCardNumber;eRFID[iPodglad].bFormPresent;eRFID[iPodglad].bBottlePresent;eRFID[iPodglad].bWeighed;
;eRFID[iPodglad].bWeightOK;
;eRFID[iPodglad].bDosed;
;eRFID[iPodglad].bCapOK;
;eRFID[iPodglad].bCapCorrectCapOn;
;eRFID[iPodglad].bCapCorrectNOK;
;eRFID[iPodglad].bCapGripperScrewed;
;eRFID[iPodglad].bCapGripperScrewAborted;
;eRFID[iPodglad].bROPPPuttedChecked;
;eRFID[iPodglad].bROPPPutted;
;eRFID[iPodglad].bROPPCapped;
;eRFID[iPodglad].bROPPCappingAborted;
;eRFID[iPodglad].tROPPCappingTime;
;eRFID[iPodglad].bROPPCappingOK;
;eRFID[iPodglad].bROPPCappingChecked;
;eRFID[iPodglad].bCapSorterPutted;
;eRFID[iPodglad].bCapSorterPuttedAborted;
END_ACTION

ACTION aStatisticsROPP:

eUnderROPPPackageState[1].bROPPPuttedChecked;
eUnderROPPPackageState[1].bROPPPutted;
eUnderROPPPackageState[1].bROPPCapped;
eUnderROPPPackageState[1].bROPPCappingAborted;
eUnderROPPPackageState[1].tROPPCappingTime;
eUnderROPPPackageState[1].bROPPCappingOK;
eUnderROPPPackageState[1].bROPPCappingChecked;

eBeforeROPPCapControlPackageState[1].nID; eBeforeROPPCapControlPackageState[1].nCardNumber; eBeforeROPPCapControlPackageState[1].bFormPresent;eBeforeROPPCapControlPackageState[1].bBottlePresent;eBeforeROPPCapControlPackageState[1].bROPPPuttedChecked;	eBeforeROPPCapControlPackageState[1].bROPPPutted;

// [1..12] Strukura przed ROPP
eBeforeROPP2PackageState[3].nID; eBeforeROPP2PackageState[3].nCardNumber; eBeforeROPP2PackageState[3].bFormPresent; eBeforeROPP2PackageState[3].bBottlePresent;	eBeforeROPP2PackageState[3].bROPPPuttedChecked;	eBeforeROPP2PackageState[3].bROPPPutted;		 eBeforeROPP2PackageState[3].bDosingTwoPhases; eBeforeROPP2PackageState[3].lrDoseVolumeSV; eBeforeROPP2PackageState[3].lrDoseVolumeSVSecondPhase;  eBeforeROPP2PackageState[3].lrDoseVolumeCV; eBeforeROPP2PackageState[3].lrDoseVolumeCVSecondPhase; eBeforeROPP2PackageState[3].nDispencerNr; eBeforeROPP2PackageState[3].nDispencerNrSecondPhase; eBeforeROPP2PackageState[3].tDispencingTime; eBeforeROPP2PackageState[3].tDispencingTimeSecondPhase; eBeforeROPP2PackageState[3].bWeighed; eBeforeROPP2PackageState[2].bWeightOK; eBeforeROPP2PackageState[3].lrWeightSV; eBeforeROPP2PackageState[3].lrWeightMeasuredCV; eBeforeROPP2PackageState[3].lrWeightCV; eBeforeROPP2PackageState[3].bCapChecked;
eBeforeROPP2PackageState[2].nID; eBeforeROPP2PackageState[2].nCardNumber; eBeforeROPP2PackageState[2].bFormPresent; eBeforeROPP2PackageState[2].bBottlePresent;	eBeforeROPP2PackageState[2].bROPPPuttedChecked;	eBeforeROPP2PackageState[2].bROPPPutted;		 eBeforeROPP2PackageState[2].bDosingTwoPhases; eBeforeROPP2PackageState[2].lrDoseVolumeSV; eBeforeROPP2PackageState[2].lrDoseVolumeSVSecondPhase;  eBeforeROPP2PackageState[2].lrDoseVolumeCV; eBeforeROPP2PackageState[2].lrDoseVolumeCVSecondPhase; eBeforeROPP2PackageState[2].nDispencerNr; eBeforeROPP2PackageState[2].nDispencerNrSecondPhase; eBeforeROPP2PackageState[2].tDispencingTime; eBeforeROPP2PackageState[2].tDispencingTimeSecondPhase; eBeforeROPP2PackageState[2].bWeighed; eBeforeROPP2PackageState[2].bWeightOK; eBeforeROPP2PackageState[2].lrWeightSV; eBeforeROPP2PackageState[2].lrWeightMeasuredCV; eBeforeROPP2PackageState[2].lrWeightCV; eBeforeROPP2PackageState[2].bCapChecked;
eBeforeROPP2PackageState[1].nID; eBeforeROPP2PackageState[1].nCardNumber; eBeforeROPP2PackageState[1].bFormPresent; eBeforeROPP2PackageState[1].bBottlePresent;	eBeforeROPP2PackageState[1].bROPPPuttedChecked;	eBeforeROPP2PackageState[1].bROPPPutted;		 eBeforeROPP2PackageState[1].bDosingTwoPhases; eBeforeROPP2PackageState[1].lrDoseVolumeSV; eBeforeROPP2PackageState[1].lrDoseVolumeSVSecondPhase;  eBeforeROPP2PackageState[1].lrDoseVolumeCV; eBeforeROPP2PackageState[1].lrDoseVolumeCVSecondPhase; eBeforeROPP2PackageState[1].nDispencerNr; eBeforeROPP2PackageState[1].nDispencerNrSecondPhase; eBeforeROPP2PackageState[1].tDispencingTime; eBeforeROPP2PackageState[1].tDispencingTimeSecondPhase; eBeforeROPP2PackageState[1].bWeighed; eBeforeROPP2PackageState[1].bWeightOK; eBeforeROPP2PackageState[1].lrWeightSV; eBeforeROPP2PackageState[1].lrWeightMeasuredCV; eBeforeROPP2PackageState[1].lrWeightCV; eBeforeROPP2PackageState[1].bCapChecked;
eBeforeROPPPackageState[2].nID;  eBeforeROPPPackageState[2].nCardNumber;  eBeforeROPPPackageState[2].bFormPresent;  eBeforeROPPPackageState[2].bBottlePresent;	eBeforeROPPPackageState[2].bROPPPuttedChecked;	eBeforeROPPPackageState[2].bROPPPutted;		 eBeforeROPPPackageState[2].bDosingTwoPhases; eBeforeROPPPackageState[2].lrDoseVolumeSV; eBeforeROPPPackageState[2].lrDoseVolumeSVSecondPhase;  eBeforeROPPPackageState[2].lrDoseVolumeCV; eBeforeROPPPackageState[2].lrDoseVolumeCVSecondPhase; eBeforeROPPPackageState[2].nDispencerNr; eBeforeROPPPackageState[2].nDispencerNrSecondPhase; eBeforeROPPPackageState[2].tDispencingTime; eBeforeROPPPackageState[2].tDispencingTimeSecondPhase; eBeforeROPPPackageState[2].bWeighed; eBeforeROPPPackageState[2].bWeightOK; eBeforeROPPPackageState[2].lrWeightSV; eBeforeROPPPackageState[2].lrWeightMeasuredCV; eBeforeROPPPackageState[2].lrWeightCV; eBeforeROPPPackageState[2].bCapChecked;
eBeforeROPPPackageState[1].nID;  eBeforeROPPPackageState[1].nCardNumber;  eBeforeROPPPackageState[1].bFormPresent;  eBeforeROPPPackageState[1].bBottlePresent;	eBeforeROPPPackageState[1].bROPPPuttedChecked;	eBeforeROPPPackageState[1].bROPPPutted;		 eBeforeROPPPackageState[1].bDosingTwoPhases; eBeforeROPPPackageState[1].lrDoseVolumeSV; eBeforeROPPPackageState[1].lrDoseVolumeSVSecondPhase;  eBeforeROPPPackageState[1].lrDoseVolumeCV; eBeforeROPPPackageState[1].lrDoseVolumeCVSecondPhase; eBeforeROPPPackageState[1].nDispencerNr; eBeforeROPPPackageState[1].nDispencerNrSecondPhase; eBeforeROPPPackageState[1].tDispencingTime; eBeforeROPPPackageState[1].tDispencingTimeSecondPhase; eBeforeROPPPackageState[1].bWeighed; eBeforeROPPPackageState[1].bWeightOK; eBeforeROPPPackageState[1].lrWeightSV; eBeforeROPPPackageState[1].lrWeightMeasuredCV; eBeforeROPPPackageState[1].lrWeightCV; eBeforeROPPPackageState[1].bCapChecked;
				
//[1..3] Struktura pod ROPP
eUnderROPPPackageState[2].nID; eUnderROPPPackageState[2].nCardNumber; eUnderROPPPackageState[2].bFormPresent; eUnderROPPPackageState[2].bBottlePresent; eUnderROPPPackageState[2].bROPPPuttedChecked; eUnderROPPPackageState[2].bROPPPutted; eUnderROPPPackageState[2].bROPPCappingAborted; eUnderROPPPackageState[2].bROPPCapped; eUnderROPPPackageState[2].bDosingTwoPhases; eUnderROPPPackageState[2].lrDoseVolumeSV; eUnderROPPPackageState[2].lrDoseVolumeSVSecondPhase;  eUnderROPPPackageState[2].lrDoseVolumeCV; eUnderROPPPackageState[2].lrDoseVolumeCVSecondPhase; eUnderROPPPackageState[2].nDispencerNr; eUnderROPPPackageState[2].nDispencerNrSecondPhase; eUnderROPPPackageState[2].tDispencingTime; eUnderROPPPackageState[2].tDispencingTimeSecondPhase; eUnderROPPPackageState[2].bWeighed; eUnderROPPPackageState[2].bWeightOK; eUnderROPPPackageState[12].lrWeightSV; eUnderROPPPackageState[2].lrWeightMeasuredCV; eUnderROPPPackageState[2].lrWeightCV; 
eUnderROPPPackageState[1].nID; eUnderROPPPackageState[1].nCardNumber; eUnderROPPPackageState[1].bFormPresent; eUnderROPPPackageState[1].bBottlePresent; eUnderROPPPackageState[1].bROPPPuttedChecked; eUnderROPPPackageState[1].bROPPPutted; eUnderROPPPackageState[1].bROPPCappingAborted; eUnderROPPPackageState[1].bROPPCapped; eUnderROPPPackageState[1].bDosingTwoPhases; eUnderROPPPackageState[1].lrDoseVolumeSV; eUnderROPPPackageState[1].lrDoseVolumeSVSecondPhase;  eUnderROPPPackageState[1].lrDoseVolumeCV; eUnderROPPPackageState[1].lrDoseVolumeCVSecondPhase; eUnderROPPPackageState[1].nDispencerNr; eUnderROPPPackageState[1].nDispencerNrSecondPhase; eUnderROPPPackageState[1].tDispencingTime; eUnderROPPPackageState[1].tDispencingTimeSecondPhase; eUnderROPPPackageState[1].bWeighed; eUnderROPPPackageState[1].bWeightOK; eUnderROPPPackageState[12].lrWeightSV; eUnderROPPPackageState[1].lrWeightMeasuredCV; eUnderROPPPackageState[1].lrWeightCV; 

//[1..2] Struktura za ROPP
eUnderROPPCorrectCapPackageState[1].nID;eUnderROPPCorrectCapPackageState[1].nCardNumber; 	eUnderROPPCorrectCapPackageState[1].bFormPresent; eUnderROPPCorrectCapPackageState[1].bBottlePresent; eUnderROPPCorrectCapPackageState[1].bROPPPuttedChecked; eUnderROPPCorrectCapPackageState[1].bROPPPutted;eUnderROPPCorrectCapPackageState[1].bROPPCappingAborted; eUnderROPPCorrectCapPackageState[1].bROPPCapped; eUnderROPPCorrectCapPackageState[1].bDosingTwoPhases; eUnderROPPCorrectCapPackageState[1].lrDoseVolumeSV; eUnderROPPCorrectCapPackageState[1].lrDoseVolumeSVSecondPhase;  eUnderCorrectCapPackageState[1].lrDoseVolumeCV; eUnderCorrectCapPackageState[1].lrDoseVolumeCVSecondPhase; eUnderROPPCorrectCapPackageState[8].nDispencerNr; eUnderROPPCorrectCapPackageState[1].nDispencerNrSecondPhase; eUnderROPPCorrectCapPackageState[1].tDispencingTime; eUnderROPPCorrectCapPackageState[1].tDispencingTimeSecondPhase; eUnderROPPCorrectCapPackageState[1].bWeighed; eUnderROPPCorrectCapPackageState[1].bWeightOK; eUnderCorrectCapPackageState[1].lrWeightSV; eUnderCorrectCapPackageState[1].lrWeightMeasuredCV; eUnderCorrectCapPackageState[1].lrWeightCV; 
										eUnderROPPCorrectCapPackageState[1].bROPPCappingOK;	eUnderROPPCorrectCapPackageState[1].bROPPCappingChecked;
										
										
eRFID[1].nCardNumber; eRFID[1].bROPPPuttedChecked;	eRFID[1].bROPPPutted;		eRFID[1].bROPPCapped;		eRFID[1].bROPPCappingAborted; eRFID[1].bROPPCappingOK;  eRFID[1].bROPPCappingChecked;eRFID[1].bFormPresent; eRFID[1].bBottlePresent; eRFID[1].bDosingTwoPhases; eRFID[1].nDispencerNr; eRFID[1].nDispencerNrSecondPhase; eRFID[1].lrDoseVolumeSV; eRFID[1].lrDoseVolumeCV; eRFID[1].lrDoseVolumeSVSecondPhase; eRFID[1].lrDoseVolumeCVSecondPhase;			eRFID[1].bDosed; 	eRFID[1].bDoseAborted; eRFID[1].bWeighed; eRFID[1].lrWeightSV; eRFID[1].lrWeightCV; eRFID[1].lrWeightMeasuredCV; eRFID[1].bWeightOK; eRFID[1].bCapPutted; eRFID[1].bCapChecked; eRFID[1].bCapOK; eRFID[1].bCapGripperScrewed; eRFID[1].bCapGripperScrewAborted; eRFID[1].bBottleTransferedToExit; eRFID[1].bBottleTransferedToLabeler;  eRFID[1].lrWeightDif; eRFID[1].lrMinWeightCV; eRFID[1].lrMaxWeightCV;
eRFID[2].nCardNumber; eRFID[2].bROPPPuttedChecked;	eRFID[2].bROPPPutted;		eRFID[2].bROPPCapped;		eRFID[2].bROPPCappingAborted; eRFID[2].bROPPCappingOK;  eRFID[2].bROPPCappingChecked;eRFID[2].bFormPresent; eRFID[2].bBottlePresent; eRFID[2].bDosingTwoPhases; eRFID[2].nDispencerNr; eRFID[2].nDispencerNrSecondPhase; eRFID[2].lrDoseVolumeSV; eRFID[2].lrDoseVolumeCV; eRFID[2].lrDoseVolumeSVSecondPhase; eRFID[2].lrDoseVolumeCVSecondPhase;			eRFID[2].bDosed; 	eRFID[2].bDoseAborted; eRFID[2].bWeighed; eRFID[2].lrWeightSV; eRFID[2].lrWeightCV; eRFID[2].lrWeightMeasuredCV; eRFID[2].bWeightOK; eRFID[2].bCapPutted; eRFID[2].bCapChecked; eRFID[2].bCapOK; eRFID[2].bCapGripperScrewed; eRFID[2].bCapGripperScrewAborted; eRFID[2].bBottleTransferedToExit; eRFID[2].bBottleTransferedToLabeler;  eRFID[2].lrWeightDif; eRFID[2].lrMinWeightCV; eRFID[2].lrMaxWeightCV;
eRFID[3].nCardNumber; eRFID[3].bROPPPuttedChecked;	eRFID[3].bROPPPutted;		eRFID[3].bROPPCapped;		eRFID[3].bROPPCappingAborted; eRFID[3].bROPPCappingOK;  eRFID[3].bROPPCappingChecked;eRFID[3].bFormPresent; eRFID[3].bBottlePresent; eRFID[3].bDosingTwoPhases; eRFID[3].nDispencerNr; eRFID[3].nDispencerNrSecondPhase; eRFID[3].lrDoseVolumeSV; eRFID[3].lrDoseVolumeCV; eRFID[3].lrDoseVolumeSVSecondPhase; eRFID[3].lrDoseVolumeCVSecondPhase;			eRFID[3].bDosed; 	eRFID[3].bDoseAborted; eRFID[3].bWeighed; eRFID[3].lrWeightSV; eRFID[3].lrWeightCV; eRFID[3].lrWeightMeasuredCV; eRFID[3].bWeightOK; eRFID[3].bCapPutted; eRFID[3].bCapChecked; eRFID[3].bCapOK; eRFID[3].bCapGripperScrewed; eRFID[3].bCapGripperScrewAborted; eRFID[3].bBottleTransferedToExit; eRFID[3].bBottleTransferedToLabeler;  eRFID[3].lrWeightDif; eRFID[3].lrMinWeightCV; eRFID[3].lrMaxWeightCV;
eRFID[4].nCardNumber; eRFID[4].bROPPPuttedChecked;	eRFID[4].bROPPPutted;		eRFID[4].bROPPCapped;		eRFID[4].bROPPCappingAborted; eRFID[4].bROPPCappingOK;  eRFID[4].bROPPCappingChecked;eRFID[4].bFormPresent; eRFID[4].bBottlePresent; eRFID[4].bDosingTwoPhases; eRFID[4].nDispencerNr; eRFID[4].nDispencerNrSecondPhase; eRFID[4].lrDoseVolumeSV; eRFID[4].lrDoseVolumeCV; eRFID[4].lrDoseVolumeSVSecondPhase; eRFID[4].lrDoseVolumeCVSecondPhase;			eRFID[4].bDosed; 	eRFID[4].bDoseAborted; eRFID[4].bWeighed; eRFID[4].lrWeightSV; eRFID[4].lrWeightCV; eRFID[4].lrWeightMeasuredCV; eRFID[4].bWeightOK; eRFID[4].bCapPutted; eRFID[4].bCapChecked; eRFID[4].bCapOK; eRFID[4].bCapGripperScrewed; eRFID[4].bCapGripperScrewAborted; eRFID[4].bBottleTransferedToExit; eRFID[4].bBottleTransferedToLabeler;  eRFID[4].lrWeightDif; eRFID[4].lrMinWeightCV; eRFID[4].lrMaxWeightCV;
eRFID[5].nCardNumber; eRFID[5].bROPPPuttedChecked;	eRFID[5].bROPPPutted;		eRFID[5].bROPPCapped;		eRFID[5].bROPPCappingAborted; eRFID[5].bROPPCappingOK;  eRFID[5].bROPPCappingChecked;eRFID[5].bFormPresent; eRFID[5].bBottlePresent; eRFID[5].bDosingTwoPhases; eRFID[5].nDispencerNr; eRFID[5].nDispencerNrSecondPhase; eRFID[5].lrDoseVolumeSV; eRFID[5].lrDoseVolumeCV; eRFID[5].lrDoseVolumeSVSecondPhase; eRFID[5].lrDoseVolumeCVSecondPhase;			eRFID[5].bDosed; 	eRFID[5].bDoseAborted; eRFID[5].bWeighed; eRFID[5].lrWeightSV; eRFID[5].lrWeightCV; eRFID[5].lrWeightMeasuredCV; eRFID[5].bWeightOK; eRFID[5].bCapPutted; eRFID[5].bCapChecked; eRFID[5].bCapOK; eRFID[5].bCapGripperScrewed; eRFID[5].bCapGripperScrewAborted; eRFID[5].bBottleTransferedToExit; eRFID[5].bBottleTransferedToLabeler;  eRFID[5].lrWeightDif; eRFID[5].lrMinWeightCV; eRFID[5].lrMaxWeightCV;
eRFID[6].nCardNumber; eRFID[6].bROPPPuttedChecked;	eRFID[6].bROPPPutted;		eRFID[6].bROPPCapped;		eRFID[6].bROPPCappingAborted; eRFID[6].bROPPCappingOK;  eRFID[6].bROPPCappingChecked;eRFID[6].bFormPresent; eRFID[6].bBottlePresent; eRFID[6].bDosingTwoPhases; eRFID[6].nDispencerNr; eRFID[6].nDispencerNrSecondPhase; eRFID[6].lrDoseVolumeSV; eRFID[6].lrDoseVolumeCV; eRFID[6].lrDoseVolumeSVSecondPhase; eRFID[6].lrDoseVolumeCVSecondPhase;			eRFID[6].bDosed; 	eRFID[6].bDoseAborted; eRFID[6].bWeighed; eRFID[6].lrWeightSV; eRFID[6].lrWeightCV; eRFID[6].lrWeightMeasuredCV; eRFID[6].bWeightOK; eRFID[6].bCapPutted; eRFID[6].bCapChecked; eRFID[6].bCapOK; eRFID[6].bCapGripperScrewed; eRFID[6].bCapGripperScrewAborted; eRFID[6].bBottleTransferedToExit; eRFID[6].bBottleTransferedToLabeler;  eRFID[6].lrWeightDif; eRFID[6].lrMinWeightCV; eRFID[6].lrMaxWeightCV;
eRFID[7].nCardNumber; eRFID[7].bROPPPuttedChecked;	eRFID[7].bROPPPutted;		eRFID[7].bROPPCapped;		eRFID[7].bROPPCappingAborted; eRFID[7].bROPPCappingOK;  eRFID[7].bROPPCappingChecked;eRFID[7].bFormPresent; eRFID[7].bBottlePresent; eRFID[7].bDosingTwoPhases; eRFID[7].nDispencerNr; eRFID[7].nDispencerNrSecondPhase; eRFID[7].lrDoseVolumeSV; eRFID[7].lrDoseVolumeCV; eRFID[7].lrDoseVolumeSVSecondPhase; eRFID[7].lrDoseVolumeCVSecondPhase;			eRFID[7].bDosed; 	eRFID[7].bDoseAborted; eRFID[7].bWeighed; eRFID[7].lrWeightSV; eRFID[7].lrWeightCV; eRFID[7].lrWeightMeasuredCV; eRFID[7].bWeightOK; eRFID[7].bCapPutted; eRFID[7].bCapChecked; eRFID[7].bCapOK; eRFID[7].bCapGripperScrewed; eRFID[7].bCapGripperScrewAborted; eRFID[7].bBottleTransferedToExit; eRFID[7].bBottleTransferedToLabeler;  eRFID[7].lrWeightDif; eRFID[7].lrMinWeightCV; eRFID[7].lrMaxWeightCV;
eRFID[8].nCardNumber; eRFID[8].bROPPPuttedChecked;	eRFID[8].bROPPPutted;		eRFID[8].bROPPCapped;		eRFID[8].bROPPCappingAborted; eRFID[8].bROPPCappingOK;  eRFID[8].bROPPCappingChecked;eRFID[8].bFormPresent; eRFID[8].bBottlePresent; eRFID[8].bDosingTwoPhases; eRFID[8].nDispencerNr; eRFID[8].nDispencerNrSecondPhase; eRFID[8].lrDoseVolumeSV; eRFID[8].lrDoseVolumeCV; eRFID[8].lrDoseVolumeSVSecondPhase; eRFID[8].lrDoseVolumeCVSecondPhase; 			eRFID[8].bDosed; 	eRFID[8].bDoseAborted; eRFID[8].bWeighed; eRFID[8].lrWeightSV; eRFID[8].lrWeightCV; eRFID[8].lrWeightMeasuredCV; eRFID[8].bWeightOK; eRFID[8].bCapPutted; eRFID[8].bCapChecked; eRFID[8].bCapOK; eRFID[8].bCapGripperScrewed; eRFID[8].bCapGripperScrewAborted; eRFID[8].bBottleTransferedToExit; eRFID[8].bBottleTransferedToLabeler;  eRFID[8].lrWeightDif; eRFID[8].lrMinWeightCV; eRFID[8].lrMaxWeightCV;
eRFID[9].nCardNumber; eRFID[9].bROPPPuttedChecked;	eRFID[9].bROPPPutted;		eRFID[9].bROPPCapped;		eRFID[9].bROPPCappingAborted; eRFID[9].bROPPCappingOK;  eRFID[9].bROPPCappingChecked;eRFID[9].bFormPresent; eRFID[9].bBottlePresent; eRFID[9].bDosingTwoPhases; eRFID[9].nDispencerNr; eRFID[9].nDispencerNrSecondPhase; eRFID[9].lrDoseVolumeSV; eRFID[9].lrDoseVolumeCV; eRFID[9].lrDoseVolumeSVSecondPhase; eRFID[9].lrDoseVolumeCVSecondPhase; 			eRFID[9].bDosed; 	eRFID[9].bDoseAborted; eRFID[9].bWeighed; eRFID[9].lrWeightSV; eRFID[9].lrWeightCV; eRFID[9].lrWeightMeasuredCV; eRFID[9].bWeightOK; eRFID[9].bCapPutted; eRFID[9].bCapChecked; eRFID[9].bCapOK; eRFID[9].bCapGripperScrewed; eRFID[9].bCapGripperScrewAborted; eRFID[9].bBottleTransferedToExit; eRFID[9].bBottleTransferedToLabeler;  eRFID[9].lrWeightDif; eRFID[9].lrMinWeightCV; eRFID[9].lrMaxWeightCV;
eRFID[10].nCardNumber;eRFID[10].bROPPPuttedChecked;	eRFID[10].bROPPPutted;		eRFID[10].bROPPCapped;		eRFID[10].bROPPCappingAborted;eRFID[10].bROPPCappingOK; eRFID[10].bROPPCappingChecked;eRFID[10].bFormPresent; eRFID[10].bBottlePresent; eRFID[10].bDosingTwoPhases; eRFID[10].nDispencerNr; eRFID[10].nDispencerNrSecondPhase; eRFID[10].lrDoseVolumeSV; eRFID[10].lrDoseVolumeCV; eRFID[10].lrDoseVolumeSVSecondPhase; eRFID[10].lrDoseVolumeCVSecondPhase; eRFID[10].bDosed;	eRFID[10].bDoseAborted; eRFID[10].bWeighed; eRFID[10].lrWeightSV; eRFID[10].lrWeightCV; eRFID[10].lrWeightMeasuredCV; eRFID[10].bWeightOK; eRFID[10].bCapPutted; eRFID[10].bCapChecked; eRFID[10].bCapOK; eRFID[10].bCapGripperScrewed; eRFID[10].bCapGripperScrewAborted; eRFID[10].bBottleTransferedToExit; eRFID[10].bBottleTransferedToLabeler; eRFID[10].lrWeightDif; eRFID[10].lrMinWeightCV;eRFID[10].lrMaxWeightCV;
eRFID[11].nCardNumber;eRFID[11].bROPPPuttedChecked;	eRFID[11].bROPPPutted;		eRFID[11].bROPPCapped;		eRFID[11].bROPPCappingAborted;eRFID[11].bROPPCappingOK; eRFID[11].bROPPCappingChecked;eRFID[11].bFormPresent; eRFID[11].bBottlePresent; eRFID[11].bDosingTwoPhases; eRFID[11].nDispencerNr; eRFID[11].nDispencerNrSecondPhase; eRFID[11].lrDoseVolumeSV; eRFID[11].lrDoseVolumeCV; eRFID[11].lrDoseVolumeSVSecondPhase; eRFID[11].lrDoseVolumeCVSecondPhase; eRFID[11].bDosed;	eRFID[11].bDoseAborted; eRFID[11].bWeighed; eRFID[11].lrWeightSV; eRFID[11].lrWeightCV; eRFID[11].lrWeightMeasuredCV; eRFID[11].bWeightOK; eRFID[11].bCapPutted; eRFID[11].bCapChecked; eRFID[11].bCapOK; eRFID[11].bCapGripperScrewed; eRFID[11].bCapGripperScrewAborted; eRFID[11].bBottleTransferedToExit; eRFID[11].bBottleTransferedToLabeler; eRFID[11].lrWeightDif; eRFID[11].lrMinWeightCV;eRFID[11].lrMaxWeightCV;
eRFID[12].nCardNumber;eRFID[12].bROPPPuttedChecked;	eRFID[12].bROPPPutted;		eRFID[12].bROPPCapped;		eRFID[12].bROPPCappingAborted;eRFID[12].bROPPCappingOK; eRFID[12].bROPPCappingChecked;eRFID[12].bFormPresent; eRFID[12].bBottlePresent; eRFID[12].bDosingTwoPhases; eRFID[12].nDispencerNr; eRFID[12].nDispencerNrSecondPhase; eRFID[12].lrDoseVolumeSV; eRFID[12].lrDoseVolumeCV; eRFID[12].lrDoseVolumeSVSecondPhase; eRFID[12].lrDoseVolumeCVSecondPhase; eRFID[12].bDosed;	eRFID[12].bDoseAborted; eRFID[12].bWeighed; eRFID[12].lrWeightSV; eRFID[12].lrWeightCV; eRFID[12].lrWeightMeasuredCV; eRFID[12].bWeightOK; eRFID[12].bCapPutted; eRFID[12].bCapChecked; eRFID[12].bCapOK; eRFID[12].bCapGripperScrewed; eRFID[12].bCapGripperScrewAborted; eRFID[12].bBottleTransferedToExit; eRFID[12].bBottleTransferedToLabeler; eRFID[12].lrWeightDif; eRFID[12].lrMinWeightCV;eRFID[12].lrMaxWeightCV;
eRFID[13].nCardNumber;eRFID[13].bROPPPuttedChecked;	eRFID[13].bROPPPutted;		eRFID[13].bROPPCapped;		eRFID[13].bROPPCappingAborted;eRFID[13].bROPPCappingOK; eRFID[13].bROPPCappingChecked;eRFID[13].bFormPresent; eRFID[13].bBottlePresent; eRFID[13].bDosingTwoPhases; eRFID[13].nDispencerNr; eRFID[13].nDispencerNrSecondPhase; eRFID[13].lrDoseVolumeSV; eRFID[13].lrDoseVolumeCV; eRFID[13].lrDoseVolumeSVSecondPhase; eRFID[13].lrDoseVolumeCVSecondPhase; eRFID[13].bDosed;	eRFID[13].bDoseAborted; eRFID[13].bWeighed; eRFID[13].lrWeightSV; eRFID[13].lrWeightCV; eRFID[13].lrWeightMeasuredCV; eRFID[13].bWeightOK; eRFID[13].bCapPutted; eRFID[13].bCapChecked; eRFID[13].bCapOK; eRFID[13].bCapGripperScrewed; eRFID[13].bCapGripperScrewAborted; eRFID[13].bBottleTransferedToExit; eRFID[13].bBottleTransferedToLabeler; eRFID[13].lrWeightDif; eRFID[13].lrMinWeightCV;eRFID[13].lrMaxWeightCV;
eRFID[14].nCardNumber;eRFID[14].bROPPPuttedChecked;	eRFID[14].bROPPPutted;		eRFID[14].bROPPCapped;		eRFID[14].bROPPCappingAborted;eRFID[14].bROPPCappingOK; eRFID[14].bROPPCappingChecked;eRFID[14].bFormPresent; eRFID[14].bBottlePresent; eRFID[14].bDosingTwoPhases; eRFID[14].nDispencerNr; eRFID[14].nDispencerNrSecondPhase; eRFID[14].lrDoseVolumeSV; eRFID[14].lrDoseVolumeCV; eRFID[14].lrDoseVolumeSVSecondPhase; eRFID[14].lrDoseVolumeCVSecondPhase; eRFID[14].bDosed;	eRFID[14].bDoseAborted; eRFID[14].bWeighed; eRFID[14].lrWeightSV; eRFID[14].lrWeightCV; eRFID[14].lrWeightMeasuredCV; eRFID[14].bWeightOK; eRFID[14].bCapPutted; eRFID[14].bCapChecked; eRFID[14].bCapOK; eRFID[14].bCapGripperScrewed; eRFID[14].bCapGripperScrewAborted; eRFID[14].bBottleTransferedToExit; eRFID[14].bBottleTransferedToLabeler; eRFID[14].lrWeightDif; eRFID[14].lrMinWeightCV;eRFID[14].lrMaxWeightCV;
eRFID[15].nCardNumber;eRFID[15].bROPPPuttedChecked;	eRFID[15].bROPPPutted;		eRFID[15].bROPPCapped;		eRFID[15].bROPPCappingAborted;eRFID[15].bROPPCappingOK; eRFID[15].bROPPCappingChecked;eRFID[15].bFormPresent; eRFID[15].bBottlePresent; eRFID[15].bDosingTwoPhases; eRFID[15].nDispencerNr; eRFID[15].nDispencerNrSecondPhase; eRFID[15].lrDoseVolumeSV; eRFID[15].lrDoseVolumeCV; eRFID[15].lrDoseVolumeSVSecondPhase; eRFID[15].lrDoseVolumeCVSecondPhase; eRFID[15].bDosed;	eRFID[15].bDoseAborted; eRFID[15].bWeighed; eRFID[15].lrWeightSV; eRFID[15].lrWeightCV; eRFID[15].lrWeightMeasuredCV; eRFID[15].bWeightOK; eRFID[15].bCapPutted; eRFID[15].bCapChecked; eRFID[15].bCapOK; eRFID[15].bCapGripperScrewed; eRFID[15].bCapGripperScrewAborted; eRFID[15].bBottleTransferedToExit; eRFID[15].bBottleTransferedToLabeler; eRFID[15].lrWeightDif; eRFID[15].lrMinWeightCV;eRFID[15].lrMaxWeightCV;
eRFID[16].nCardNumber;eRFID[16].bROPPPuttedChecked;	eRFID[16].bROPPPutted;		eRFID[16].bROPPCapped;		eRFID[16].bROPPCappingAborted;eRFID[16].bROPPCappingOK; eRFID[16].bROPPCappingChecked;eRFID[16].bFormPresent; eRFID[16].bBottlePresent; eRFID[16].bDosingTwoPhases; eRFID[16].nDispencerNr; eRFID[16].nDispencerNrSecondPhase; eRFID[16].lrDoseVolumeSV; eRFID[16].lrDoseVolumeCV; eRFID[16].lrDoseVolumeSVSecondPhase; eRFID[16].lrDoseVolumeCVSecondPhase; eRFID[16].bDosed;	eRFID[16].bDoseAborted; eRFID[16].bWeighed; eRFID[16].lrWeightSV; eRFID[16].lrWeightCV; eRFID[16].lrWeightMeasuredCV; eRFID[16].bWeightOK; eRFID[16].bCapPutted; eRFID[16].bCapChecked; eRFID[16].bCapOK; eRFID[16].bCapGripperScrewed; eRFID[16].bCapGripperScrewAborted; eRFID[16].bBottleTransferedToExit; eRFID[16].bBottleTransferedToLabeler; eRFID[16].lrWeightDif; eRFID[16].lrMinWeightCV;eRFID[16].lrMaxWeightCV;
eRFID[17].nCardNumber;eRFID[17].bROPPPuttedChecked;	eRFID[17].bROPPPutted;		eRFID[17].bROPPCapped;		eRFID[17].bROPPCappingAborted;eRFID[17].bROPPCappingOK; eRFID[17].bROPPCappingChecked;eRFID[17].bFormPresent; eRFID[17].bBottlePresent; eRFID[17].bDosingTwoPhases; eRFID[17].nDispencerNr; eRFID[17].nDispencerNrSecondPhase; eRFID[17].lrDoseVolumeSV; eRFID[17].lrDoseVolumeCV; eRFID[17].lrDoseVolumeSVSecondPhase; eRFID[17].lrDoseVolumeCVSecondPhase; eRFID[17].bDosed;	eRFID[17].bDoseAborted; eRFID[17].bWeighed; eRFID[17].lrWeightSV; eRFID[17].lrWeightCV; eRFID[17].lrWeightMeasuredCV; eRFID[17].bWeightOK; eRFID[17].bCapPutted; eRFID[17].bCapChecked; eRFID[17].bCapOK; eRFID[17].bCapGripperScrewed; eRFID[17].bCapGripperScrewAborted; eRFID[17].bBottleTransferedToExit; eRFID[17].bBottleTransferedToLabeler; eRFID[17].lrWeightDif; eRFID[17].lrMinWeightCV;eRFID[17].lrMaxWeightCV;
eRFID[18].nCardNumber;eRFID[18].bROPPPuttedChecked;	eRFID[18].bROPPPutted;		eRFID[18].bROPPCapped;		eRFID[18].bROPPCappingAborted;eRFID[18].bROPPCappingOK; eRFID[18].bROPPCappingChecked;eRFID[18].bFormPresent; eRFID[18].bBottlePresent; eRFID[18].bDosingTwoPhases; eRFID[18].nDispencerNr; eRFID[18].nDispencerNrSecondPhase; eRFID[18].lrDoseVolumeSV; eRFID[18].lrDoseVolumeCV; eRFID[18].lrDoseVolumeSVSecondPhase; eRFID[18].lrDoseVolumeCVSecondPhase; eRFID[18].bDosed;	eRFID[18].bDoseAborted; eRFID[18].bWeighed; eRFID[18].lrWeightSV; eRFID[18].lrWeightCV; eRFID[18].lrWeightMeasuredCV; eRFID[18].bWeightOK; eRFID[18].bCapPutted; eRFID[18].bCapChecked; eRFID[18].bCapOK; eRFID[18].bCapGripperScrewed; eRFID[18].bCapGripperScrewAborted; eRFID[18].bBottleTransferedToExit; eRFID[18].bBottleTransferedToLabeler; eRFID[18].lrWeightDif; eRFID[18].lrMinWeightCV;eRFID[18].lrMaxWeightCV;
eRFID[19].nCardNumber;eRFID[19].bROPPPuttedChecked;	eRFID[19].bROPPPutted;		eRFID[19].bROPPCapped;		eRFID[19].bROPPCappingAborted;eRFID[19].bROPPCappingOK; eRFID[19].bROPPCappingChecked;eRFID[19].bFormPresent; eRFID[19].bBottlePresent; eRFID[19].bDosingTwoPhases; eRFID[19].nDispencerNr; eRFID[19].nDispencerNrSecondPhase; eRFID[19].lrDoseVolumeSV; eRFID[19].lrDoseVolumeCV; eRFID[19].lrDoseVolumeSVSecondPhase; eRFID[19].lrDoseVolumeCVSecondPhase; eRFID[19].bDosed;	eRFID[19].bDoseAborted; eRFID[19].bWeighed; eRFID[19].lrWeightSV; eRFID[19].lrWeightCV; eRFID[19].lrWeightMeasuredCV; eRFID[19].bWeightOK; eRFID[19].bCapPutted; eRFID[19].bCapChecked; eRFID[19].bCapOK; eRFID[19].bCapGripperScrewed; eRFID[19].bCapGripperScrewAborted; eRFID[19].bBottleTransferedToExit; eRFID[19].bBottleTransferedToLabeler; eRFID[19].lrWeightDif; eRFID[19].lrMinWeightCV;eRFID[19].lrMaxWeightCV;
eRFID[20].nCardNumber;eRFID[20].bROPPPuttedChecked;	eRFID[20].bROPPPutted;		eRFID[20].bROPPCapped;		eRFID[20].bROPPCappingAborted;eRFID[20].bROPPCappingOK; eRFID[20].bROPPCappingChecked;eRFID[20].bFormPresent; eRFID[20].bBottlePresent; eRFID[20].bDosingTwoPhases; eRFID[20].nDispencerNr; eRFID[20].nDispencerNrSecondPhase; eRFID[20].lrDoseVolumeSV; eRFID[20].lrDoseVolumeCV; eRFID[20].lrDoseVolumeSVSecondPhase; eRFID[20].lrDoseVolumeCVSecondPhase; eRFID[20].bDosed;	eRFID[20].bDoseAborted; eRFID[20].bWeighed; eRFID[20].lrWeightSV; eRFID[20].lrWeightCV; eRFID[20].lrWeightMeasuredCV; eRFID[20].bWeightOK; eRFID[20].bCapPutted; eRFID[20].bCapChecked; eRFID[20].bCapOK; eRFID[20].bCapGripperScrewed; eRFID[20].bCapGripperScrewAborted; eRFID[20].bBottleTransferedToExit; eRFID[20].bBottleTransferedToLabeler; eRFID[20].lrWeightDif; eRFID[20].lrMinWeightCV;eRFID[20].lrMaxWeightCV;
eRFID[21].nCardNumber;eRFID[21].bROPPPuttedChecked;	eRFID[21].bROPPPutted;		eRFID[21].bROPPCapped;		eRFID[21].bROPPCappingAborted;eRFID[21].bROPPCappingOK; eRFID[21].bROPPCappingChecked;eRFID[21].bFormPresent; eRFID[21].bBottlePresent; eRFID[21].bDosingTwoPhases; eRFID[21].nDispencerNr; eRFID[21].nDispencerNrSecondPhase; eRFID[21].lrDoseVolumeSV; eRFID[21].lrDoseVolumeCV; eRFID[21].lrDoseVolumeSVSecondPhase; eRFID[21].lrDoseVolumeCVSecondPhase; eRFID[21].bDosed;	eRFID[21].bDoseAborted; eRFID[21].bWeighed; eRFID[21].lrWeightSV; eRFID[21].lrWeightCV; eRFID[21].lrWeightMeasuredCV; eRFID[21].bWeightOK; eRFID[21].bCapPutted; eRFID[21].bCapChecked; eRFID[21].bCapOK; eRFID[21].bCapGripperScrewed; eRFID[21].bCapGripperScrewAborted; eRFID[21].bBottleTransferedToExit; eRFID[21].bBottleTransferedToLabeler; eRFID[21].lrWeightDif; eRFID[21].lrMinWeightCV;eRFID[21].lrMaxWeightCV;
eRFID[22].nCardNumber;eRFID[22].bROPPPuttedChecked;	eRFID[22].bROPPPutted;		eRFID[22].bROPPCapped;		eRFID[22].bROPPCappingAborted;eRFID[22].bROPPCappingOK; eRFID[22].bROPPCappingChecked;eRFID[22].bFormPresent; eRFID[22].bBottlePresent; eRFID[22].bDosingTwoPhases; eRFID[22].nDispencerNr; eRFID[22].nDispencerNrSecondPhase; eRFID[22].lrDoseVolumeSV; eRFID[22].lrDoseVolumeCV; eRFID[22].lrDoseVolumeSVSecondPhase; eRFID[22].lrDoseVolumeCVSecondPhase; eRFID[22].bDosed;	eRFID[22].bDoseAborted; eRFID[22].bWeighed; eRFID[22].lrWeightSV; eRFID[22].lrWeightCV; eRFID[22].lrWeightMeasuredCV; eRFID[22].bWeightOK; eRFID[22].bCapPutted; eRFID[22].bCapChecked; eRFID[22].bCapOK; eRFID[22].bCapGripperScrewed; eRFID[22].bCapGripperScrewAborted; eRFID[22].bBottleTransferedToExit; eRFID[22].bBottleTransferedToLabeler; eRFID[22].lrWeightDif; eRFID[22].lrMinWeightCV;eRFID[22].lrMaxWeightCV;
eRFID[23].nCardNumber;eRFID[23].bROPPPuttedChecked;	eRFID[23].bROPPPutted;		eRFID[23].bROPPCapped;		eRFID[23].bROPPCappingAborted;eRFID[23].bROPPCappingOK; eRFID[23].bROPPCappingChecked;eRFID[23].bFormPresent; eRFID[23].bBottlePresent; eRFID[23].bDosingTwoPhases; eRFID[23].nDispencerNr; eRFID[23].nDispencerNrSecondPhase; eRFID[23].lrDoseVolumeSV; eRFID[23].lrDoseVolumeCV; eRFID[23].lrDoseVolumeSVSecondPhase; eRFID[23].lrDoseVolumeCVSecondPhase; eRFID[23].bDosed;	eRFID[23].bDoseAborted; eRFID[23].bWeighed; eRFID[23].lrWeightSV; eRFID[23].lrWeightCV; eRFID[23].lrWeightMeasuredCV; eRFID[23].bWeightOK; eRFID[23].bCapPutted; eRFID[23].bCapChecked; eRFID[23].bCapOK; eRFID[23].bCapGripperScrewed; eRFID[23].bCapGripperScrewAborted; eRFID[23].bBottleTransferedToExit; eRFID[23].bBottleTransferedToLabeler; eRFID[23].lrWeightDif; eRFID[23].lrMinWeightCV;eRFID[23].lrMaxWeightCV;
eRFID[24].nCardNumber;eRFID[24].bROPPPuttedChecked;	eRFID[24].bROPPPutted;		eRFID[24].bROPPCapped;		eRFID[24].bROPPCappingAborted;eRFID[24].bROPPCappingOK; eRFID[24].bROPPCappingChecked;eRFID[24].bFormPresent; eRFID[24].bBottlePresent; eRFID[24].bDosingTwoPhases; eRFID[24].nDispencerNr; eRFID[24].nDispencerNrSecondPhase; eRFID[24].lrDoseVolumeSV; eRFID[24].lrDoseVolumeCV; eRFID[24].lrDoseVolumeSVSecondPhase; eRFID[24].lrDoseVolumeCVSecondPhase; eRFID[24].bDosed;	eRFID[24].bDoseAborted; eRFID[24].bWeighed; eRFID[24].lrWeightSV; eRFID[24].lrWeightCV; eRFID[24].lrWeightMeasuredCV; eRFID[24].bWeightOK; eRFID[24].bCapPutted; eRFID[24].bCapChecked; eRFID[24].bCapOK; eRFID[24].bCapGripperScrewed; eRFID[24].bCapGripperScrewAborted; eRFID[24].bBottleTransferedToExit; eRFID[24].bBottleTransferedToLabeler; eRFID[24].lrWeightDif; eRFID[24].lrMinWeightCV;eRFID[24].lrMaxWeightCV;
eRFID[25].nCardNumber;eRFID[25].bROPPPuttedChecked;	eRFID[25].bROPPPutted;		eRFID[25].bROPPCapped;		eRFID[25].bROPPCappingAborted;eRFID[25].bROPPCappingOK; eRFID[25].bROPPCappingChecked;eRFID[25].bFormPresent; eRFID[25].bBottlePresent; eRFID[25].bDosingTwoPhases; eRFID[25].nDispencerNr; eRFID[25].nDispencerNrSecondPhase; eRFID[25].lrDoseVolumeSV; eRFID[25].lrDoseVolumeCV; eRFID[25].lrDoseVolumeSVSecondPhase; eRFID[25].lrDoseVolumeCVSecondPhase; eRFID[25].bDosed;	eRFID[25].bDoseAborted; eRFID[25].bWeighed; eRFID[25].lrWeightSV; eRFID[25].lrWeightCV; eRFID[25].lrWeightMeasuredCV; eRFID[25].bWeightOK; eRFID[25].bCapPutted; eRFID[25].bCapChecked; eRFID[25].bCapOK; eRFID[25].bCapGripperScrewed; eRFID[25].bCapGripperScrewAborted; eRFID[25].bBottleTransferedToExit; eRFID[25].bBottleTransferedToLabeler; eRFID[25].lrWeightDif; eRFID[25].lrMinWeightCV;eRFID[25].lrMaxWeightCV;
eRFID[26].nCardNumber;eRFID[26].bROPPPuttedChecked;	eRFID[26].bROPPPutted;		eRFID[26].bROPPCapped;		eRFID[26].bROPPCappingAborted;eRFID[26].bROPPCappingOK; eRFID[26].bROPPCappingChecked;eRFID[26].bFormPresent; eRFID[26].bBottlePresent; eRFID[26].bDosingTwoPhases; eRFID[26].nDispencerNr; eRFID[26].nDispencerNrSecondPhase; eRFID[26].lrDoseVolumeSV; eRFID[26].lrDoseVolumeCV; eRFID[26].lrDoseVolumeSVSecondPhase; eRFID[26].lrDoseVolumeCVSecondPhase; eRFID[26].bDosed;	eRFID[26].bDoseAborted; eRFID[26].bWeighed; eRFID[26].lrWeightSV; eRFID[26].lrWeightCV; eRFID[26].lrWeightMeasuredCV; eRFID[26].bWeightOK; eRFID[26].bCapPutted; eRFID[26].bCapChecked; eRFID[26].bCapOK; eRFID[26].bCapGripperScrewed; eRFID[26].bCapGripperScrewAborted; eRFID[26].bBottleTransferedToExit; eRFID[26].bBottleTransferedToLabeler; eRFID[26].lrWeightDif; eRFID[26].lrMinWeightCV;eRFID[26].lrMaxWeightCV;
eRFID[27].nCardNumber;eRFID[27].bROPPPuttedChecked;	eRFID[27].bROPPPutted;		eRFID[27].bROPPCapped;		eRFID[27].bROPPCappingAborted;eRFID[27].bROPPCappingOK; eRFID[27].bROPPCappingChecked;eRFID[27].bFormPresent; eRFID[27].bBottlePresent; eRFID[27].bDosingTwoPhases; eRFID[27].nDispencerNr; eRFID[27].nDispencerNrSecondPhase; eRFID[27].lrDoseVolumeSV; eRFID[27].lrDoseVolumeCV; eRFID[27].lrDoseVolumeSVSecondPhase; eRFID[27].lrDoseVolumeCVSecondPhase; eRFID[27].bDosed;	eRFID[27].bDoseAborted; eRFID[27].bWeighed; eRFID[27].lrWeightSV; eRFID[27].lrWeightCV; eRFID[27].lrWeightMeasuredCV; eRFID[27].bWeightOK; eRFID[27].bCapPutted; eRFID[27].bCapChecked; eRFID[27].bCapOK; eRFID[27].bCapGripperScrewed; eRFID[27].bCapGripperScrewAborted; eRFID[27].bBottleTransferedToExit; eRFID[27].bBottleTransferedToLabeler; eRFID[27].lrWeightDif; eRFID[27].lrMinWeightCV;eRFID[27].lrMaxWeightCV;
eRFID[28].nCardNumber;eRFID[28].bROPPPuttedChecked;	eRFID[28].bROPPPutted;		eRFID[28].bROPPCapped;		eRFID[28].bROPPCappingAborted;eRFID[28].bROPPCappingOK; eRFID[28].bROPPCappingChecked;eRFID[28].bFormPresent; eRFID[28].bBottlePresent; eRFID[28].bDosingTwoPhases; eRFID[28].nDispencerNr; eRFID[28].nDispencerNrSecondPhase; eRFID[28].lrDoseVolumeSV; eRFID[28].lrDoseVolumeCV; eRFID[28].lrDoseVolumeSVSecondPhase; eRFID[28].lrDoseVolumeCVSecondPhase; eRFID[28].bDosed;	eRFID[28].bDoseAborted; eRFID[28].bWeighed; eRFID[28].lrWeightSV; eRFID[28].lrWeightCV; eRFID[28].lrWeightMeasuredCV; eRFID[28].bWeightOK; eRFID[28].bCapPutted; eRFID[28].bCapChecked; eRFID[28].bCapOK; eRFID[28].bCapGripperScrewed; eRFID[28].bCapGripperScrewAborted; eRFID[28].bBottleTransferedToExit; eRFID[28].bBottleTransferedToLabeler; eRFID[28].lrWeightDif; eRFID[28].lrMinWeightCV;eRFID[28].lrMaxWeightCV;
eRFID[29].nCardNumber;eRFID[29].bROPPPuttedChecked;	eRFID[29].bROPPPutted;		eRFID[29].bROPPCapped;		eRFID[29].bROPPCappingAborted;eRFID[29].bROPPCappingOK; eRFID[29].bROPPCappingChecked;eRFID[29].bFormPresent; eRFID[29].bBottlePresent; eRFID[29].bDosingTwoPhases; eRFID[29].nDispencerNr; eRFID[29].nDispencerNrSecondPhase; eRFID[29].lrDoseVolumeSV; eRFID[29].lrDoseVolumeCV; eRFID[29].lrDoseVolumeSVSecondPhase; eRFID[29].lrDoseVolumeCVSecondPhase;	eRFID[29].bDosed;	eRFID[29].bDoseAborted; eRFID[29].bWeighed; eRFID[29].lrWeightSV; eRFID[29].lrWeightCV; eRFID[29].lrWeightMeasuredCV; eRFID[29].bWeightOK; eRFID[29].bCapPutted; eRFID[29].bCapChecked; eRFID[29].bCapOK; eRFID[29].bCapGripperScrewed; eRFID[29].bCapGripperScrewAborted; eRFID[29].bBottleTransferedToExit; eRFID[29].bBottleTransferedToLabeler; eRFID[29].lrWeightDif; eRFID[29].lrMinWeightCV;eRFID[29].lrMaxWeightCV;
eRFID[30].nCardNumber;eRFID[30].bROPPPuttedChecked;	eRFID[30].bROPPPutted;		eRFID[30].bROPPCapped;		eRFID[30].bROPPCappingAborted;eRFID[30].bROPPCappingOK; eRFID[30].bROPPCappingChecked;eRFID[30].bFormPresent; eRFID[30].bBottlePresent; eRFID[30].bDosingTwoPhases; eRFID[30].nDispencerNr; eRFID[30].nDispencerNrSecondPhase; eRFID[30].lrDoseVolumeSV; eRFID[30].lrDoseVolumeCV; eRFID[30].lrDoseVolumeSVSecondPhase; eRFID[30].lrDoseVolumeCVSecondPhase;	eRFID[30].bDosed;	eRFID[30].bDoseAborted; eRFID[30].bWeighed; eRFID[30].lrWeightSV; eRFID[30].lrWeightCV; eRFID[30].lrWeightMeasuredCV; eRFID[30].bWeightOK; eRFID[30].bCapPutted; eRFID[30].bCapChecked; eRFID[30].bCapOK; eRFID[30].bCapGripperScrewed; eRFID[30].bCapGripperScrewAborted; eRFID[30].bBottleTransferedToExit; eRFID[30].bBottleTransferedToLabeler; eRFID[30].lrWeightDif; eRFID[30].lrMinWeightCV;eRFID[30].lrMaxWeightCV;
eRFID[31].nCardNumber;eRFID[31].bROPPPuttedChecked;	eRFID[31].bROPPPutted;		eRFID[31].bROPPCapped;		eRFID[31].bROPPCappingAborted;eRFID[31].bROPPCappingOK; eRFID[31].bROPPCappingChecked;eRFID[31].bFormPresent; eRFID[31].bBottlePresent; eRFID[31].bDosingTwoPhases; eRFID[31].nDispencerNr; eRFID[31].nDispencerNrSecondPhase; eRFID[31].lrDoseVolumeSV; eRFID[31].lrDoseVolumeCV; eRFID[31].lrDoseVolumeSVSecondPhase; eRFID[31].lrDoseVolumeCVSecondPhase;	eRFID[31].bDosed;	eRFID[31].bDoseAborted; eRFID[31].bWeighed; eRFID[31].lrWeightSV; eRFID[31].lrWeightCV; eRFID[31].lrWeightMeasuredCV; eRFID[31].bWeightOK; eRFID[31].bCapPutted; eRFID[31].bCapChecked; eRFID[31].bCapOK; eRFID[31].bCapGripperScrewed; eRFID[31].bCapGripperScrewAborted; eRFID[31].bBottleTransferedToExit; eRFID[31].bBottleTransferedToLabeler; eRFID[31].lrWeightDif; eRFID[31].lrMinWeightCV;eRFID[31].lrMaxWeightCV;
eRFID[32].nCardNumber;eRFID[32].bROPPPuttedChecked;	eRFID[32].bROPPPutted;		eRFID[32].bROPPCapped;		eRFID[32].bROPPCappingAborted;eRFID[32].bROPPCappingOK; eRFID[32].bROPPCappingChecked;eRFID[32].bFormPresent; eRFID[32].bBottlePresent; eRFID[32].bDosingTwoPhases; eRFID[32].nDispencerNr; eRFID[32].nDispencerNrSecondPhase; eRFID[32].lrDoseVolumeSV; eRFID[32].lrDoseVolumeCV; eRFID[32].lrDoseVolumeSVSecondPhase; eRFID[32].lrDoseVolumeCVSecondPhase;	eRFID[32].bDosed;	eRFID[32].bDoseAborted; eRFID[32].bWeighed; eRFID[32].lrWeightSV; eRFID[32].lrWeightCV; eRFID[32].lrWeightMeasuredCV; eRFID[32].bWeightOK; eRFID[32].bCapPutted; eRFID[32].bCapChecked; eRFID[32].bCapOK; eRFID[32].bCapGripperScrewed; eRFID[32].bCapGripperScrewAborted; eRFID[32].bBottleTransferedToExit; eRFID[32].bBottleTransferedToLabeler; eRFID[32].lrWeightDif; eRFID[32].lrMinWeightCV;eRFID[32].lrMaxWeightCV;
eRFID[33].nCardNumber;eRFID[33].bROPPPuttedChecked;	eRFID[33].bROPPPutted;		eRFID[33].bROPPCapped;		eRFID[33].bROPPCappingAborted;eRFID[33].bROPPCappingOK; eRFID[33].bROPPCappingChecked;eRFID[33].bFormPresent; eRFID[33].bBottlePresent; eRFID[33].bDosingTwoPhases; eRFID[33].nDispencerNr; eRFID[33].nDispencerNrSecondPhase; eRFID[33].lrDoseVolumeSV; eRFID[33].lrDoseVolumeCV; eRFID[33].lrDoseVolumeSVSecondPhase; eRFID[33].lrDoseVolumeCVSecondPhase;	eRFID[33].bDosed;	eRFID[33].bDoseAborted; eRFID[33].bWeighed; eRFID[33].lrWeightSV; eRFID[33].lrWeightCV; eRFID[33].lrWeightMeasuredCV; eRFID[33].bWeightOK; eRFID[33].bCapPutted; eRFID[33].bCapChecked; eRFID[33].bCapOK; eRFID[33].bCapGripperScrewed; eRFID[33].bCapGripperScrewAborted; eRFID[33].bBottleTransferedToExit; eRFID[33].bBottleTransferedToLabeler; eRFID[33].lrWeightDif; eRFID[33].lrMinWeightCV;eRFID[33].lrMaxWeightCV;
eRFID[34].nCardNumber;eRFID[34].bROPPPuttedChecked;	eRFID[34].bROPPPutted;		eRFID[34].bROPPCapped;		eRFID[34].bROPPCappingAborted;eRFID[34].bROPPCappingOK; eRFID[34].bROPPCappingChecked;eRFID[34].bFormPresent; eRFID[34].bBottlePresent; eRFID[34].bDosingTwoPhases; eRFID[34].nDispencerNr; eRFID[34].nDispencerNrSecondPhase; eRFID[34].lrDoseVolumeSV; eRFID[34].lrDoseVolumeCV; eRFID[34].lrDoseVolumeSVSecondPhase; eRFID[34].lrDoseVolumeCVSecondPhase;	eRFID[34].bDosed;	eRFID[34].bDoseAborted; eRFID[34].bWeighed; eRFID[34].lrWeightSV; eRFID[34].lrWeightCV; eRFID[34].lrWeightMeasuredCV; eRFID[34].bWeightOK; eRFID[34].bCapPutted; eRFID[34].bCapChecked; eRFID[34].bCapOK; eRFID[34].bCapGripperScrewed; eRFID[34].bCapGripperScrewAborted; eRFID[34].bBottleTransferedToExit; eRFID[34].bBottleTransferedToLabeler; eRFID[34].lrWeightDif; eRFID[34].lrMinWeightCV;eRFID[34].lrMaxWeightCV;
eRFID[35].nCardNumber;eRFID[35].bROPPPuttedChecked;	eRFID[35].bROPPPutted;		eRFID[35].bROPPCapped;		eRFID[35].bROPPCappingAborted;eRFID[35].bROPPCappingOK; eRFID[35].bROPPCappingChecked;eRFID[35].bFormPresent; eRFID[35].bBottlePresent; eRFID[35].bDosingTwoPhases; eRFID[35].nDispencerNr; eRFID[35].nDispencerNrSecondPhase; eRFID[35].lrDoseVolumeSV; eRFID[35].lrDoseVolumeCV; eRFID[35].lrDoseVolumeSVSecondPhase; eRFID[35].lrDoseVolumeCVSecondPhase;	eRFID[35].bDosed;	eRFID[35].bDoseAborted; eRFID[35].bWeighed; eRFID[35].lrWeightSV; eRFID[35].lrWeightCV; eRFID[35].lrWeightMeasuredCV; eRFID[35].bWeightOK; eRFID[35].bCapPutted; eRFID[35].bCapChecked; eRFID[35].bCapOK; eRFID[35].bCapGripperScrewed; eRFID[35].bCapGripperScrewAborted; eRFID[35].bBottleTransferedToExit; eRFID[35].bBottleTransferedToLabeler; eRFID[35].lrWeightDif; eRFID[35].lrMinWeightCV;eRFID[35].lrMaxWeightCV;
eRFID[36].nCardNumber;eRFID[36].bROPPPuttedChecked;	eRFID[36].bROPPPutted;		eRFID[36].bROPPCapped;		eRFID[36].bROPPCappingAborted;eRFID[36].bROPPCappingOK; eRFID[36].bROPPCappingChecked;eRFID[36].bFormPresent; eRFID[36].bBottlePresent; eRFID[36].bDosingTwoPhases; eRFID[36].nDispencerNr; eRFID[36].nDispencerNrSecondPhase; eRFID[36].lrDoseVolumeSV; eRFID[36].lrDoseVolumeCV; eRFID[36].lrDoseVolumeSVSecondPhase; eRFID[36].lrDoseVolumeCVSecondPhase;	eRFID[36].bDosed;	eRFID[36].bDoseAborted; eRFID[36].bWeighed; eRFID[36].lrWeightSV; eRFID[36].lrWeightCV; eRFID[36].lrWeightMeasuredCV; eRFID[36].bWeightOK; eRFID[36].bCapPutted; eRFID[36].bCapChecked; eRFID[36].bCapOK; eRFID[36].bCapGripperScrewed; eRFID[36].bCapGripperScrewAborted; eRFID[36].bBottleTransferedToExit; eRFID[36].bBottleTransferedToLabeler; eRFID[36].lrWeightDif; eRFID[36].lrMinWeightCV;eRFID[36].lrMaxWeightCV;
eRFID[37].nCardNumber;eRFID[37].bROPPPuttedChecked;	eRFID[37].bROPPPutted;		eRFID[37].bROPPCapped;		eRFID[37].bROPPCappingAborted;eRFID[37].bROPPCappingOK; eRFID[37].bROPPCappingChecked;eRFID[37].bFormPresent; eRFID[37].bBottlePresent; eRFID[37].bDosingTwoPhases; eRFID[37].nDispencerNr; eRFID[37].nDispencerNrSecondPhase; eRFID[37].lrDoseVolumeSV; eRFID[37].lrDoseVolumeCV; eRFID[37].lrDoseVolumeSVSecondPhase; eRFID[37].lrDoseVolumeCVSecondPhase;	eRFID[37].bDosed;	eRFID[37].bDoseAborted; eRFID[37].bWeighed; eRFID[37].lrWeightSV; eRFID[37].lrWeightCV; eRFID[37].lrWeightMeasuredCV; eRFID[37].bWeightOK; eRFID[37].bCapPutted; eRFID[37].bCapChecked; eRFID[37].bCapOK; eRFID[37].bCapGripperScrewed; eRFID[37].bCapGripperScrewAborted; eRFID[37].bBottleTransferedToExit; eRFID[37].bBottleTransferedToLabeler; eRFID[37].lrWeightDif; eRFID[37].lrMinWeightCV;eRFID[37].lrMaxWeightCV;
eRFID[38].nCardNumber;eRFID[38].bROPPPuttedChecked;	eRFID[38].bROPPPutted;		eRFID[38].bROPPCapped;		eRFID[38].bROPPCappingAborted;eRFID[38].bROPPCappingOK; eRFID[38].bROPPCappingChecked;eRFID[38].bFormPresent; eRFID[38].bBottlePresent; eRFID[38].bDosingTwoPhases; eRFID[38].nDispencerNr; eRFID[38].nDispencerNrSecondPhase; eRFID[38].lrDoseVolumeSV; eRFID[38].lrDoseVolumeCV; eRFID[38].lrDoseVolumeSVSecondPhase; eRFID[38].lrDoseVolumeCVSecondPhase;	eRFID[38].bDosed;	eRFID[38].bDoseAborted; eRFID[38].bWeighed; eRFID[38].lrWeightSV; eRFID[38].lrWeightCV; eRFID[38].lrWeightMeasuredCV; eRFID[38].bWeightOK; eRFID[38].bCapPutted; eRFID[38].bCapChecked; eRFID[38].bCapOK; eRFID[38].bCapGripperScrewed; eRFID[38].bCapGripperScrewAborted; eRFID[38].bBottleTransferedToExit; eRFID[38].bBottleTransferedToLabeler; eRFID[38].lrWeightDif; eRFID[38].lrMinWeightCV;eRFID[38].lrMaxWeightCV;
eRFID[39].nCardNumber;eRFID[39].bROPPPuttedChecked;	eRFID[39].bROPPPutted;		eRFID[39].bROPPCapped;		eRFID[39].bROPPCappingAborted;eRFID[39].bROPPCappingOK; eRFID[39].bROPPCappingChecked;eRFID[39].bFormPresent; eRFID[39].bBottlePresent; eRFID[39].bDosingTwoPhases; eRFID[39].nDispencerNr; eRFID[39].nDispencerNrSecondPhase; eRFID[39].lrDoseVolumeSV; eRFID[39].lrDoseVolumeCV; eRFID[39].lrDoseVolumeSVSecondPhase; eRFID[39].lrDoseVolumeCVSecondPhase;	eRFID[39].bDosed;	eRFID[39].bDoseAborted; eRFID[39].bWeighed; eRFID[39].lrWeightSV; eRFID[39].lrWeightCV; eRFID[39].lrWeightMeasuredCV; eRFID[39].bWeightOK; eRFID[39].bCapPutted; eRFID[39].bCapChecked; eRFID[39].bCapOK; eRFID[39].bCapGripperScrewed; eRFID[39].bCapGripperScrewAborted; eRFID[39].bBottleTransferedToExit; eRFID[39].bBottleTransferedToLabeler; eRFID[39].lrWeightDif; eRFID[39].lrMinWeightCV;eRFID[39].lrMaxWeightCV;
eRFID[40].nCardNumber;eRFID[40].bROPPPuttedChecked;	eRFID[40].bROPPPutted;		eRFID[40].bROPPCapped;		eRFID[40].bROPPCappingAborted;eRFID[40].bROPPCappingOK; eRFID[40].bROPPCappingChecked;eRFID[40].bFormPresent; eRFID[40].bBottlePresent; eRFID[40].bDosingTwoPhases; eRFID[40].nDispencerNr; eRFID[40].nDispencerNrSecondPhase; eRFID[40].lrDoseVolumeSV; eRFID[40].lrDoseVolumeCV; eRFID[40].lrDoseVolumeSVSecondPhase; eRFID[40].lrDoseVolumeCVSecondPhase;	eRFID[40].bDosed;	eRFID[40].bDoseAborted; eRFID[40].bWeighed; eRFID[40].lrWeightSV; eRFID[40].lrWeightCV; eRFID[40].lrWeightMeasuredCV; eRFID[40].bWeightOK; eRFID[40].bCapPutted; eRFID[40].bCapChecked; eRFID[40].bCapOK; eRFID[40].bCapGripperScrewed; eRFID[40].bCapGripperScrewAborted; eRFID[40].bBottleTransferedToExit; eRFID[40].bBottleTransferedToLabeler; eRFID[40].lrWeightDif; eRFID[40].lrMinWeightCV;eRFID[40].lrMaxWeightCV;
eRFID[41].nCardNumber;eRFID[41].bROPPPuttedChecked;	eRFID[41].bROPPPutted;		eRFID[41].bROPPCapped;		eRFID[41].bROPPCappingAborted;eRFID[41].bROPPCappingOK; eRFID[41].bROPPCappingChecked;eRFID[41].bFormPresent; eRFID[41].bBottlePresent; eRFID[41].bDosingTwoPhases; eRFID[41].nDispencerNr; eRFID[41].nDispencerNrSecondPhase; eRFID[41].lrDoseVolumeSV; eRFID[41].lrDoseVolumeCV; eRFID[41].lrDoseVolumeSVSecondPhase; eRFID[41].lrDoseVolumeCVSecondPhase;	eRFID[41].bDosed;	eRFID[41].bDoseAborted; eRFID[41].bWeighed; eRFID[41].lrWeightSV; eRFID[41].lrWeightCV; eRFID[41].lrWeightMeasuredCV; eRFID[41].bWeightOK; eRFID[41].bCapPutted; eRFID[41].bCapChecked; eRFID[41].bCapOK; eRFID[41].bCapGripperScrewed; eRFID[41].bCapGripperScrewAborted; eRFID[41].bBottleTransferedToExit; eRFID[41].bBottleTransferedToLabeler; eRFID[41].lrWeightDif; eRFID[41].lrMinWeightCV;eRFID[41].lrMaxWeightCV;
eRFID[42].nCardNumber;eRFID[42].bROPPPuttedChecked;	eRFID[42].bROPPPutted;		eRFID[42].bROPPCapped;		eRFID[42].bROPPCappingAborted;eRFID[42].bROPPCappingOK; eRFID[42].bROPPCappingChecked;eRFID[42].bFormPresent; eRFID[42].bBottlePresent; eRFID[42].bDosingTwoPhases; eRFID[42].nDispencerNr; eRFID[42].nDispencerNrSecondPhase; eRFID[42].lrDoseVolumeSV; eRFID[42].lrDoseVolumeCV; eRFID[42].lrDoseVolumeSVSecondPhase; eRFID[42].lrDoseVolumeCVSecondPhase;	eRFID[42].bDosed;	eRFID[42].bDoseAborted; eRFID[42].bWeighed; eRFID[42].lrWeightSV; eRFID[42].lrWeightCV; eRFID[42].lrWeightMeasuredCV; eRFID[42].bWeightOK; eRFID[42].bCapPutted; eRFID[42].bCapChecked; eRFID[42].bCapOK; eRFID[42].bCapGripperScrewed; eRFID[42].bCapGripperScrewAborted; eRFID[42].bBottleTransferedToExit; eRFID[42].bBottleTransferedToLabeler; eRFID[42].lrWeightDif; eRFID[42].lrMinWeightCV;eRFID[42].lrMaxWeightCV;
eRFID[43].nCardNumber;eRFID[43].bROPPPuttedChecked;	eRFID[43].bROPPPutted;		eRFID[43].bROPPCapped;		eRFID[43].bROPPCappingAborted;eRFID[43].bROPPCappingOK; eRFID[43].bROPPCappingChecked;eRFID[43].bFormPresent; eRFID[43].bBottlePresent; eRFID[43].bDosingTwoPhases; eRFID[43].nDispencerNr; eRFID[43].nDispencerNrSecondPhase; eRFID[43].lrDoseVolumeSV; eRFID[43].lrDoseVolumeCV; eRFID[43].lrDoseVolumeSVSecondPhase; eRFID[43].lrDoseVolumeCVSecondPhase;	eRFID[43].bDosed;	eRFID[43].bDoseAborted; eRFID[43].bWeighed; eRFID[43].lrWeightSV; eRFID[43].lrWeightCV; eRFID[43].lrWeightMeasuredCV; eRFID[43].bWeightOK; eRFID[43].bCapPutted; eRFID[43].bCapChecked; eRFID[43].bCapOK; eRFID[43].bCapGripperScrewed; eRFID[43].bCapGripperScrewAborted; eRFID[43].bBottleTransferedToExit; eRFID[43].bBottleTransferedToLabeler; eRFID[43].lrWeightDif; eRFID[43].lrMinWeightCV;eRFID[43].lrMaxWeightCV;
eRFID[44].nCardNumber;eRFID[44].bROPPPuttedChecked;	eRFID[44].bROPPPutted;		eRFID[44].bROPPCapped;		eRFID[44].bROPPCappingAborted;eRFID[44].bROPPCappingOK; eRFID[44].bROPPCappingChecked;eRFID[44].bFormPresent; eRFID[44].bBottlePresent; eRFID[44].bDosingTwoPhases; eRFID[44].nDispencerNr; eRFID[44].nDispencerNrSecondPhase; eRFID[44].lrDoseVolumeSV; eRFID[44].lrDoseVolumeCV; eRFID[44].lrDoseVolumeSVSecondPhase; eRFID[44].lrDoseVolumeCVSecondPhase;	eRFID[44].bDosed;	eRFID[44].bDoseAborted; eRFID[44].bWeighed; eRFID[44].lrWeightSV; eRFID[44].lrWeightCV; eRFID[44].lrWeightMeasuredCV; eRFID[44].bWeightOK; eRFID[44].bCapPutted; eRFID[44].bCapChecked; eRFID[44].bCapOK; eRFID[44].bCapGripperScrewed; eRFID[44].bCapGripperScrewAborted; eRFID[44].bBottleTransferedToExit; eRFID[44].bBottleTransferedToLabeler; eRFID[44].lrWeightDif; eRFID[44].lrMinWeightCV;eRFID[44].lrMaxWeightCV;
eRFID[45].nCardNumber;eRFID[45].bROPPPuttedChecked;	eRFID[45].bROPPPutted;		eRFID[45].bROPPCapped;		eRFID[45].bROPPCappingAborted;eRFID[45].bROPPCappingOK; eRFID[45].bROPPCappingChecked;eRFID[45].bFormPresent; eRFID[45].bBottlePresent; eRFID[45].bDosingTwoPhases; eRFID[45].nDispencerNr; eRFID[45].nDispencerNrSecondPhase; eRFID[45].lrDoseVolumeSV; eRFID[45].lrDoseVolumeCV; eRFID[45].lrDoseVolumeSVSecondPhase; eRFID[45].lrDoseVolumeCVSecondPhase;	eRFID[45].bDosed;	eRFID[45].bDoseAborted; eRFID[45].bWeighed; eRFID[45].lrWeightSV; eRFID[45].lrWeightCV; eRFID[45].lrWeightMeasuredCV; eRFID[45].bWeightOK; eRFID[45].bCapPutted; eRFID[45].bCapChecked; eRFID[45].bCapOK; eRFID[45].bCapGripperScrewed; eRFID[45].bCapGripperScrewAborted; eRFID[45].bBottleTransferedToExit; eRFID[45].bBottleTransferedToLabeler; eRFID[45].lrWeightDif; eRFID[45].lrMinWeightCV;eRFID[45].lrMaxWeightCV;
eRFID[46].nCardNumber;eRFID[46].bROPPPuttedChecked;	eRFID[46].bROPPPutted;		eRFID[46].bROPPCapped;		eRFID[46].bROPPCappingAborted;eRFID[46].bROPPCappingOK; eRFID[46].bROPPCappingChecked;eRFID[46].bFormPresent; eRFID[46].bBottlePresent; eRFID[46].bDosingTwoPhases; eRFID[46].nDispencerNr; eRFID[46].nDispencerNrSecondPhase; eRFID[46].lrDoseVolumeSV; eRFID[46].lrDoseVolumeCV; eRFID[46].lrDoseVolumeSVSecondPhase; eRFID[46].lrDoseVolumeCVSecondPhase;	eRFID[46].bDosed;	eRFID[46].bDoseAborted; eRFID[46].bWeighed; eRFID[46].lrWeightSV; eRFID[46].lrWeightCV; eRFID[46].lrWeightMeasuredCV; eRFID[46].bWeightOK; eRFID[46].bCapPutted; eRFID[46].bCapChecked; eRFID[46].bCapOK; eRFID[46].bCapGripperScrewed; eRFID[46].bCapGripperScrewAborted; eRFID[46].bBottleTransferedToExit; eRFID[46].bBottleTransferedToLabeler; eRFID[46].lrWeightDif; eRFID[46].lrMinWeightCV;eRFID[46].lrMaxWeightCV;
eRFID[47].nCardNumber;eRFID[47].bROPPPuttedChecked;	eRFID[47].bROPPPutted;		eRFID[47].bROPPCapped;		eRFID[47].bROPPCappingAborted;eRFID[47].bROPPCappingOK; eRFID[47].bROPPCappingChecked;eRFID[47].bFormPresent; eRFID[47].bBottlePresent; eRFID[47].bDosingTwoPhases; eRFID[47].nDispencerNr; eRFID[47].nDispencerNrSecondPhase; eRFID[47].lrDoseVolumeSV; eRFID[47].lrDoseVolumeCV; eRFID[47].lrDoseVolumeSVSecondPhase; eRFID[47].lrDoseVolumeCVSecondPhase;	eRFID[47].bDosed;	eRFID[47].bDoseAborted; eRFID[47].bWeighed; eRFID[47].lrWeightSV; eRFID[47].lrWeightCV; eRFID[47].lrWeightMeasuredCV; eRFID[47].bWeightOK; eRFID[47].bCapPutted; eRFID[47].bCapChecked; eRFID[47].bCapOK; eRFID[47].bCapGripperScrewed; eRFID[47].bCapGripperScrewAborted; eRFID[47].bBottleTransferedToExit; eRFID[47].bBottleTransferedToLabeler; eRFID[47].lrWeightDif; eRFID[47].lrMinWeightCV;eRFID[47].lrMaxWeightCV;
eRFID[48].nCardNumber;eRFID[48].bROPPPuttedChecked;	eRFID[48].bROPPPutted;		eRFID[48].bROPPCapped;		eRFID[48].bROPPCappingAborted;eRFID[48].bROPPCappingOK; eRFID[48].bROPPCappingChecked;eRFID[48].bFormPresent; eRFID[48].bBottlePresent; eRFID[48].bDosingTwoPhases; eRFID[48].nDispencerNr; eRFID[48].nDispencerNrSecondPhase; eRFID[48].lrDoseVolumeSV; eRFID[48].lrDoseVolumeCV; eRFID[48].lrDoseVolumeSVSecondPhase; eRFID[48].lrDoseVolumeCVSecondPhase;	eRFID[48].bDosed;	eRFID[48].bDoseAborted; eRFID[48].bWeighed; eRFID[48].lrWeightSV; eRFID[48].lrWeightCV; eRFID[48].lrWeightMeasuredCV; eRFID[48].bWeightOK; eRFID[48].bCapPutted; eRFID[48].bCapChecked; eRFID[48].bCapOK; eRFID[48].bCapGripperScrewed; eRFID[48].bCapGripperScrewAborted; eRFID[48].bBottleTransferedToExit; eRFID[48].bBottleTransferedToLabeler; eRFID[48].lrWeightDif; eRFID[48].lrMinWeightCV;eRFID[48].lrMaxWeightCV;
eRFID[49].nCardNumber;eRFID[49].bROPPPuttedChecked;	eRFID[49].bROPPPutted;		eRFID[49].bROPPCapped;		eRFID[49].bROPPCappingAborted;eRFID[49].bROPPCappingOK; eRFID[49].bROPPCappingChecked;eRFID[49].bFormPresent; eRFID[49].bBottlePresent; eRFID[49].bDosingTwoPhases; eRFID[49].nDispencerNr; eRFID[49].nDispencerNrSecondPhase; eRFID[49].lrDoseVolumeSV; eRFID[49].lrDoseVolumeCV; eRFID[49].lrDoseVolumeSVSecondPhase; eRFID[49].lrDoseVolumeCVSecondPhase;	eRFID[49].bDosed;	eRFID[49].bDoseAborted; eRFID[49].bWeighed; eRFID[49].lrWeightSV; eRFID[49].lrWeightCV; eRFID[49].lrWeightMeasuredCV; eRFID[49].bWeightOK; eRFID[49].bCapPutted; eRFID[49].bCapChecked; eRFID[49].bCapOK; eRFID[49].bCapGripperScrewed; eRFID[49].bCapGripperScrewAborted; eRFID[49].bBottleTransferedToExit; eRFID[49].bBottleTransferedToLabeler; eRFID[49].lrWeightDif; eRFID[49].lrMinWeightCV;eRFID[49].lrMaxWeightCV;
eRFID[50].nCardNumber;eRFID[50].bROPPPuttedChecked;	eRFID[50].bROPPPutted;		eRFID[50].bROPPCapped;		eRFID[50].bROPPCappingAborted;eRFID[50].bROPPCappingOK; eRFID[50].bROPPCappingChecked;eRFID[50].bFormPresent; eRFID[50].bBottlePresent; eRFID[50].bDosingTwoPhases; eRFID[50].nDispencerNr; eRFID[50].nDispencerNrSecondPhase; eRFID[50].lrDoseVolumeSV; eRFID[50].lrDoseVolumeCV; eRFID[50].lrDoseVolumeSVSecondPhase; eRFID[50].lrDoseVolumeCVSecondPhase;	eRFID[50].bDosed;	eRFID[50].bDoseAborted; eRFID[50].bWeighed; eRFID[50].lrWeightSV; eRFID[50].lrWeightCV; eRFID[50].lrWeightMeasuredCV; eRFID[50].bWeightOK; eRFID[50].bCapPutted; eRFID[50].bCapChecked; eRFID[50].bCapOK; eRFID[50].bCapGripperScrewed; eRFID[50].bCapGripperScrewAborted; eRFID[50].bBottleTransferedToExit; eRFID[50].bBottleTransferedToLabeler; eRFID[50].lrWeightDif; eRFID[50].lrMinWeightCV;eRFID[50].lrMaxWeightCV;
eRFID[51].nCardNumber;eRFID[51].bROPPPuttedChecked;	eRFID[51].bROPPPutted;		eRFID[51].bROPPCapped;		eRFID[51].bROPPCappingAborted;eRFID[51].bROPPCappingOK; eRFID[51].bROPPCappingChecked;eRFID[51].bFormPresent; eRFID[51].bBottlePresent; eRFID[51].bDosingTwoPhases; eRFID[51].nDispencerNr; eRFID[51].nDispencerNrSecondPhase; eRFID[51].lrDoseVolumeSV; eRFID[51].lrDoseVolumeCV; eRFID[51].lrDoseVolumeSVSecondPhase; eRFID[51].lrDoseVolumeCVSecondPhase;	eRFID[51].bDosed;	eRFID[51].bDoseAborted; eRFID[51].bWeighed; eRFID[51].lrWeightSV; eRFID[51].lrWeightCV; eRFID[51].lrWeightMeasuredCV; eRFID[51].bWeightOK; eRFID[51].bCapPutted; eRFID[51].bCapChecked; eRFID[51].bCapOK; eRFID[51].bCapGripperScrewed; eRFID[51].bCapGripperScrewAborted; eRFID[51].bBottleTransferedToExit; eRFID[51].bBottleTransferedToLabeler; eRFID[51].lrWeightDif; eRFID[51].lrMinWeightCV;eRFID[51].lrMaxWeightCV;
eRFID[52].nCardNumber;eRFID[52].bROPPPuttedChecked;	eRFID[52].bROPPPutted;		eRFID[52].bROPPCapped;		eRFID[52].bROPPCappingAborted;eRFID[52].bROPPCappingOK; eRFID[52].bROPPCappingChecked;eRFID[52].bFormPresent; eRFID[52].bBottlePresent; eRFID[52].bDosingTwoPhases; eRFID[52].nDispencerNr; eRFID[52].nDispencerNrSecondPhase; eRFID[52].lrDoseVolumeSV; eRFID[52].lrDoseVolumeCV; eRFID[52].lrDoseVolumeSVSecondPhase; eRFID[52].lrDoseVolumeCVSecondPhase;	eRFID[52].bDosed;	eRFID[52].bDoseAborted; eRFID[52].bWeighed; eRFID[52].lrWeightSV; eRFID[52].lrWeightCV; eRFID[52].lrWeightMeasuredCV; eRFID[52].bWeightOK; eRFID[52].bCapPutted; eRFID[52].bCapChecked; eRFID[52].bCapOK; eRFID[52].bCapGripperScrewed; eRFID[52].bCapGripperScrewAborted; eRFID[52].bBottleTransferedToExit; eRFID[52].bBottleTransferedToLabeler; eRFID[52].lrWeightDif; eRFID[52].lrMinWeightCV;eRFID[52].lrMaxWeightCV;
eRFID[53].nCardNumber;eRFID[53].bROPPPuttedChecked;	eRFID[53].bROPPPutted;		eRFID[53].bROPPCapped;		eRFID[53].bROPPCappingAborted;eRFID[53].bROPPCappingOK; eRFID[53].bROPPCappingChecked;eRFID[53].bFormPresent; eRFID[53].bBottlePresent; eRFID[53].bDosingTwoPhases; eRFID[53].nDispencerNr; eRFID[53].nDispencerNrSecondPhase; eRFID[53].lrDoseVolumeSV; eRFID[53].lrDoseVolumeCV; eRFID[53].lrDoseVolumeSVSecondPhase; eRFID[53].lrDoseVolumeCVSecondPhase; eRFID[53].bDosed;	eRFID[53].bDoseAborted; eRFID[53].bWeighed; eRFID[53].lrWeightSV; eRFID[53].lrWeightCV; eRFID[53].lrWeightMeasuredCV; eRFID[53].bWeightOK; eRFID[53].bCapPutted; eRFID[53].bCapChecked; eRFID[53].bCapOK; eRFID[53].bCapGripperScrewed; eRFID[53].bCapGripperScrewAborted; eRFID[53].bBottleTransferedToExit; eRFID[53].bBottleTransferedToLabeler; eRFID[53].lrWeightDif; eRFID[53].lrMinWeightCV;eRFID[53].lrMaxWeightCV;
eRFID[54].nCardNumber;eRFID[54].bROPPPuttedChecked;	eRFID[54].bROPPPutted;		eRFID[54].bROPPCapped;		eRFID[54].bROPPCappingAborted;eRFID[54].bROPPCappingOK; eRFID[54].bROPPCappingChecked;eRFID[54].bFormPresent; eRFID[54].bBottlePresent; eRFID[54].bDosingTwoPhases; eRFID[54].nDispencerNr; eRFID[54].nDispencerNrSecondPhase; eRFID[54].lrDoseVolumeSV; eRFID[54].lrDoseVolumeCV; eRFID[54].lrDoseVolumeSVSecondPhase; eRFID[54].lrDoseVolumeCVSecondPhase; eRFID[54].bDosed;	eRFID[54].bDoseAborted; eRFID[54].bWeighed; eRFID[54].lrWeightSV; eRFID[54].lrWeightCV; eRFID[54].lrWeightMeasuredCV; eRFID[54].bWeightOK; eRFID[54].bCapPutted; eRFID[54].bCapChecked; eRFID[54].bCapOK; eRFID[54].bCapGripperScrewed; eRFID[54].bCapGripperScrewAborted; eRFID[54].bBottleTransferedToExit; eRFID[54].bBottleTransferedToLabeler; eRFID[54].lrWeightDif; eRFID[54].lrMinWeightCV;eRFID[54].lrMaxWeightCV;
eRFID[55].nCardNumber;eRFID[55].bROPPPuttedChecked;	eRFID[55].bROPPPutted;		eRFID[55].bROPPCapped;		eRFID[55].bROPPCappingAborted;eRFID[55].bROPPCappingOK; eRFID[55].bROPPCappingChecked;eRFID[55].bFormPresent; eRFID[55].bBottlePresent; eRFID[55].bDosingTwoPhases; eRFID[55].nDispencerNr; eRFID[55].nDispencerNrSecondPhase; eRFID[55].lrDoseVolumeSV; eRFID[55].lrDoseVolumeCV; eRFID[55].lrDoseVolumeSVSecondPhase; eRFID[55].lrDoseVolumeCVSecondPhase; eRFID[55].bDosed;	eRFID[55].bDoseAborted; eRFID[55].bWeighed; eRFID[55].lrWeightSV; eRFID[55].lrWeightCV; eRFID[55].lrWeightMeasuredCV; eRFID[55].bWeightOK; eRFID[55].bCapPutted; eRFID[55].bCapChecked; eRFID[55].bCapOK; eRFID[55].bCapGripperScrewed; eRFID[55].bCapGripperScrewAborted; eRFID[55].bBottleTransferedToExit; eRFID[55].bBottleTransferedToLabeler; eRFID[55].lrWeightDif; eRFID[55].lrMinWeightCV;eRFID[55].lrMaxWeightCV;
eRFID[56].nCardNumber;eRFID[56].bROPPPuttedChecked;	eRFID[56].bROPPPutted;		eRFID[56].bROPPCapped;		eRFID[56].bROPPCappingAborted;eRFID[56].bROPPCappingOK; eRFID[56].bROPPCappingChecked;eRFID[56].bFormPresent; eRFID[56].bBottlePresent; eRFID[56].bDosingTwoPhases; eRFID[56].nDispencerNr; eRFID[56].nDispencerNrSecondPhase; eRFID[56].lrDoseVolumeSV; eRFID[56].lrDoseVolumeCV; eRFID[56].lrDoseVolumeSVSecondPhase; eRFID[56].lrDoseVolumeCVSecondPhase; eRFID[56].bDosed;	eRFID[56].bDoseAborted; eRFID[56].bWeighed; eRFID[56].lrWeightSV; eRFID[56].lrWeightCV; eRFID[56].lrWeightMeasuredCV; eRFID[56].bWeightOK; eRFID[56].bCapPutted; eRFID[56].bCapChecked; eRFID[56].bCapOK; eRFID[56].bCapGripperScrewed; eRFID[56].bCapGripperScrewAborted; eRFID[56].bBottleTransferedToExit; eRFID[56].bBottleTransferedToLabeler; eRFID[56].lrWeightDif; eRFID[56].lrMinWeightCV;eRFID[56].lrMaxWeightCV;
eRFID[57].nCardNumber;eRFID[57].bROPPPuttedChecked;	eRFID[57].bROPPPutted;		eRFID[57].bROPPCapped;		eRFID[57].bROPPCappingAborted;eRFID[57].bROPPCappingOK; eRFID[57].bROPPCappingChecked;eRFID[57].bFormPresent; eRFID[57].bBottlePresent; eRFID[57].bDosingTwoPhases; eRFID[57].nDispencerNr; eRFID[57].nDispencerNrSecondPhase; eRFID[57].lrDoseVolumeSV; eRFID[57].lrDoseVolumeCV; eRFID[57].lrDoseVolumeSVSecondPhase; eRFID[57].lrDoseVolumeCVSecondPhase; eRFID[57].bDosed;	eRFID[57].bDoseAborted; eRFID[57].bWeighed; eRFID[57].lrWeightSV; eRFID[57].lrWeightCV; eRFID[57].lrWeightMeasuredCV; eRFID[57].bWeightOK; eRFID[57].bCapPutted; eRFID[57].bCapChecked; eRFID[57].bCapOK; eRFID[57].bCapGripperScrewed; eRFID[57].bCapGripperScrewAborted; eRFID[57].bBottleTransferedToExit; eRFID[57].bBottleTransferedToLabeler; eRFID[57].lrWeightDif; eRFID[57].lrMinWeightCV;eRFID[57].lrMaxWeightCV;
eRFID[58].nCardNumber;eRFID[58].bROPPPuttedChecked;	eRFID[58].bROPPPutted;		eRFID[58].bROPPCapped;		eRFID[58].bROPPCappingAborted;eRFID[58].bROPPCappingOK; eRFID[58].bROPPCappingChecked;eRFID[58].bFormPresent; eRFID[58].bBottlePresent; eRFID[58].bDosingTwoPhases; eRFID[58].nDispencerNr; eRFID[58].nDispencerNrSecondPhase; eRFID[58].lrDoseVolumeSV; eRFID[58].lrDoseVolumeCV; eRFID[58].lrDoseVolumeSVSecondPhase; eRFID[58].lrDoseVolumeCVSecondPhase; eRFID[58].bDosed;	eRFID[58].bDoseAborted; eRFID[58].bWeighed; eRFID[58].lrWeightSV; eRFID[58].lrWeightCV; eRFID[58].lrWeightMeasuredCV; eRFID[58].bWeightOK; eRFID[58].bCapPutted; eRFID[58].bCapChecked; eRFID[58].bCapOK; eRFID[58].bCapGripperScrewed; eRFID[58].bCapGripperScrewAborted; eRFID[58].bBottleTransferedToExit; eRFID[58].bBottleTransferedToLabeler; eRFID[58].lrWeightDif; eRFID[58].lrMinWeightCV;eRFID[58].lrMaxWeightCV;
eRFID[59].nCardNumber;eRFID[59].bROPPPuttedChecked;	eRFID[59].bROPPPutted;		eRFID[59].bROPPCapped;		eRFID[59].bROPPCappingAborted;eRFID[59].bROPPCappingOK; eRFID[59].bROPPCappingChecked;eRFID[59].bFormPresent; eRFID[59].bBottlePresent; eRFID[59].bDosingTwoPhases; eRFID[59].nDispencerNr; eRFID[59].nDispencerNrSecondPhase; eRFID[59].lrDoseVolumeSV; eRFID[59].lrDoseVolumeCV; eRFID[59].lrDoseVolumeSVSecondPhase; eRFID[59].lrDoseVolumeCVSecondPhase; eRFID[59].bDosed;	eRFID[59].bDoseAborted; eRFID[59].bWeighed; eRFID[59].lrWeightSV; eRFID[59].lrWeightCV; eRFID[59].lrWeightMeasuredCV; eRFID[59].bWeightOK; eRFID[59].bCapPutted; eRFID[59].bCapChecked; eRFID[59].bCapOK; eRFID[59].bCapGripperScrewed; eRFID[59].bCapGripperScrewAborted; eRFID[59].bBottleTransferedToExit; eRFID[59].bBottleTransferedToLabeler; eRFID[59].lrWeightDif; eRFID[59].lrMinWeightCV;eRFID[59].lrMaxWeightCV;
eRFID[60].nCardNumber;eRFID[60].bROPPPuttedChecked;	eRFID[60].bROPPPutted;		eRFID[60].bROPPCapped;		eRFID[60].bROPPCappingAborted;eRFID[60].bROPPCappingOK; eRFID[60].bROPPCappingChecked;eRFID[60].bFormPresent; eRFID[60].bBottlePresent; eRFID[60].bDosingTwoPhases; eRFID[60].nDispencerNr; eRFID[60].nDispencerNrSecondPhase; eRFID[60].lrDoseVolumeSV; eRFID[60].lrDoseVolumeCV; eRFID[60].lrDoseVolumeSVSecondPhase; eRFID[60].lrDoseVolumeCVSecondPhase; eRFID[60].bDosed;	eRFID[60].bDoseAborted; eRFID[60].bWeighed; eRFID[60].lrWeightSV; eRFID[60].lrWeightCV; eRFID[60].lrWeightMeasuredCV; eRFID[60].bWeightOK; eRFID[60].bCapPutted; eRFID[60].bCapChecked; eRFID[60].bCapOK; eRFID[60].bCapGripperScrewed; eRFID[60].bCapGripperScrewAborted; eRFID[60].bBottleTransferedToExit; eRFID[60].bBottleTransferedToLabeler; eRFID[60].lrWeightDif; eRFID[60].lrMinWeightCV;eRFID[60].lrMaxWeightCV;
eRFID[61].nCardNumber;eRFID[61].bROPPPuttedChecked;	eRFID[61].bROPPPutted;		eRFID[61].bROPPCapped;		eRFID[61].bROPPCappingAborted;eRFID[61].bROPPCappingOK; eRFID[61].bROPPCappingChecked;eRFID[61].bFormPresent; eRFID[61].bBottlePresent; eRFID[61].bDosingTwoPhases; eRFID[61].nDispencerNr; eRFID[61].nDispencerNrSecondPhase; eRFID[61].lrDoseVolumeSV; eRFID[61].lrDoseVolumeCV; eRFID[61].lrDoseVolumeSVSecondPhase; eRFID[61].lrDoseVolumeCVSecondPhase; eRFID[61].bDosed;	eRFID[61].bDoseAborted; eRFID[61].bWeighed; eRFID[61].lrWeightSV; eRFID[61].lrWeightCV; eRFID[61].lrWeightMeasuredCV; eRFID[61].bWeightOK; eRFID[61].bCapPutted; eRFID[61].bCapChecked; eRFID[61].bCapOK; eRFID[61].bCapGripperScrewed; eRFID[61].bCapGripperScrewAborted; eRFID[61].bBottleTransferedToExit; eRFID[61].bBottleTransferedToLabeler; eRFID[61].lrWeightDif; eRFID[61].lrMinWeightCV;eRFID[61].lrMaxWeightCV;
eRFID[62].nCardNumber;eRFID[62].bROPPPuttedChecked;	eRFID[62].bROPPPutted;		eRFID[62].bROPPCapped;		eRFID[62].bROPPCappingAborted;eRFID[62].bROPPCappingOK; eRFID[62].bROPPCappingChecked;eRFID[62].bFormPresent; eRFID[62].bBottlePresent; eRFID[62].bDosingTwoPhases; eRFID[62].nDispencerNr; eRFID[62].nDispencerNrSecondPhase; eRFID[62].lrDoseVolumeSV; eRFID[62].lrDoseVolumeCV; eRFID[62].lrDoseVolumeSVSecondPhase; eRFID[62].lrDoseVolumeCVSecondPhase; eRFID[62].bDosed;	eRFID[62].bDoseAborted; eRFID[62].bWeighed; eRFID[62].lrWeightSV; eRFID[62].lrWeightCV; eRFID[62].lrWeightMeasuredCV; eRFID[62].bWeightOK; eRFID[62].bCapPutted; eRFID[62].bCapChecked; eRFID[62].bCapOK; eRFID[62].bCapGripperScrewed; eRFID[62].bCapGripperScrewAborted; eRFID[62].bBottleTransferedToExit; eRFID[62].bBottleTransferedToLabeler; eRFID[62].lrWeightDif; eRFID[62].lrMinWeightCV;eRFID[62].lrMaxWeightCV;
eRFID[63].nCardNumber;eRFID[63].bROPPPuttedChecked;	eRFID[63].bROPPPutted;		eRFID[63].bROPPCapped;		eRFID[63].bROPPCappingAborted;eRFID[63].bROPPCappingOK; eRFID[63].bROPPCappingChecked;eRFID[63].bFormPresent; eRFID[63].bBottlePresent; eRFID[63].bDosingTwoPhases; eRFID[63].nDispencerNr; eRFID[63].nDispencerNrSecondPhase; eRFID[63].lrDoseVolumeSV; eRFID[63].lrDoseVolumeCV; eRFID[63].lrDoseVolumeSVSecondPhase; eRFID[63].lrDoseVolumeCVSecondPhase; eRFID[63].bDosed;	eRFID[63].bDoseAborted; eRFID[63].bWeighed; eRFID[63].lrWeightSV; eRFID[63].lrWeightCV; eRFID[63].lrWeightMeasuredCV; eRFID[63].bWeightOK; eRFID[63].bCapPutted; eRFID[63].bCapChecked; eRFID[63].bCapOK; eRFID[63].bCapGripperScrewed; eRFID[63].bCapGripperScrewAborted; eRFID[63].bBottleTransferedToExit; eRFID[63].bBottleTransferedToLabeler; eRFID[63].lrWeightDif; eRFID[63].lrMinWeightCV;eRFID[63].lrMaxWeightCV;
eRFID[64].nCardNumber;eRFID[64].bROPPPuttedChecked;	eRFID[64].bROPPPutted;		eRFID[64].bROPPCapped;		eRFID[64].bROPPCappingAborted;eRFID[64].bROPPCappingOK; eRFID[64].bROPPCappingChecked;eRFID[64].bFormPresent; eRFID[64].bBottlePresent; eRFID[64].bDosingTwoPhases; eRFID[64].nDispencerNr; eRFID[64].nDispencerNrSecondPhase; eRFID[64].lrDoseVolumeSV; eRFID[64].lrDoseVolumeCV; eRFID[64].lrDoseVolumeSVSecondPhase; eRFID[64].lrDoseVolumeCVSecondPhase; eRFID[64].bDosed;	eRFID[64].bDoseAborted; eRFID[64].bWeighed; eRFID[64].lrWeightSV; eRFID[64].lrWeightCV; eRFID[64].lrWeightMeasuredCV; eRFID[64].bWeightOK; eRFID[64].bCapPutted; eRFID[64].bCapChecked; eRFID[64].bCapOK; eRFID[64].bCapGripperScrewed; eRFID[64].bCapGripperScrewAborted; eRFID[64].bBottleTransferedToExit; eRFID[64].bBottleTransferedToLabeler; eRFID[64].lrWeightDif; eRFID[64].lrMinWeightCV;eRFID[64].lrMaxWeightCV;
eRFID[65].nCardNumber;eRFID[65].bROPPPuttedChecked;	eRFID[65].bROPPPutted;		eRFID[65].bROPPCapped;		eRFID[65].bROPPCappingAborted;eRFID[65].bROPPCappingOK; eRFID[65].bROPPCappingChecked;eRFID[65].bFormPresent; eRFID[65].bBottlePresent; eRFID[65].bDosingTwoPhases; eRFID[65].nDispencerNr; eRFID[65].nDispencerNrSecondPhase; eRFID[65].lrDoseVolumeSV; eRFID[65].lrDoseVolumeCV; eRFID[65].lrDoseVolumeSVSecondPhase; eRFID[65].lrDoseVolumeCVSecondPhase; eRFID[65].bDosed;	eRFID[65].bDoseAborted; eRFID[65].bWeighed; eRFID[65].lrWeightSV; eRFID[65].lrWeightCV; eRFID[65].lrWeightMeasuredCV; eRFID[65].bWeightOK; eRFID[65].bCapPutted; eRFID[65].bCapChecked; eRFID[65].bCapOK; eRFID[65].bCapGripperScrewed; eRFID[65].bCapGripperScrewAborted; eRFID[65].bBottleTransferedToExit; eRFID[65].bBottleTransferedToLabeler; eRFID[65].lrWeightDif; eRFID[65].lrMinWeightCV;eRFID[65].lrMaxWeightCV;
eRFID[66].nCardNumber;eRFID[66].bROPPPuttedChecked;	eRFID[66].bROPPPutted;		eRFID[66].bROPPCapped;		eRFID[66].bROPPCappingAborted;eRFID[66].bROPPCappingOK; eRFID[66].bROPPCappingChecked;eRFID[66].bFormPresent; eRFID[66].bBottlePresent; eRFID[66].bDosingTwoPhases; eRFID[66].nDispencerNr; eRFID[66].nDispencerNrSecondPhase; eRFID[66].lrDoseVolumeSV; eRFID[66].lrDoseVolumeCV; eRFID[66].lrDoseVolumeSVSecondPhase; eRFID[66].lrDoseVolumeCVSecondPhase; eRFID[66].bDosed;	eRFID[66].bDoseAborted; eRFID[66].bWeighed; eRFID[66].lrWeightSV; eRFID[66].lrWeightCV; eRFID[66].lrWeightMeasuredCV; eRFID[66].bWeightOK; eRFID[66].bCapPutted; eRFID[66].bCapChecked; eRFID[66].bCapOK; eRFID[66].bCapGripperScrewed; eRFID[66].bCapGripperScrewAborted; eRFID[66].bBottleTransferedToExit; eRFID[66].bBottleTransferedToLabeler; eRFID[66].lrWeightDif; eRFID[66].lrMinWeightCV;eRFID[66].lrMaxWeightCV;
eRFID[67].nCardNumber;eRFID[67].bROPPPuttedChecked;	eRFID[67].bROPPPutted;		eRFID[67].bROPPCapped;		eRFID[67].bROPPCappingAborted;eRFID[67].bROPPCappingOK; eRFID[67].bROPPCappingChecked;eRFID[67].bFormPresent; eRFID[67].bBottlePresent; eRFID[67].bDosingTwoPhases; eRFID[67].nDispencerNr; eRFID[67].nDispencerNrSecondPhase; eRFID[67].lrDoseVolumeSV; eRFID[67].lrDoseVolumeCV; eRFID[67].lrDoseVolumeSVSecondPhase; eRFID[67].lrDoseVolumeCVSecondPhase; eRFID[67].bDosed;	eRFID[67].bDoseAborted; eRFID[67].bWeighed; eRFID[67].lrWeightSV; eRFID[67].lrWeightCV; eRFID[67].lrWeightMeasuredCV; eRFID[67].bWeightOK; eRFID[67].bCapPutted; eRFID[67].bCapChecked; eRFID[67].bCapOK; eRFID[67].bCapGripperScrewed; eRFID[67].bCapGripperScrewAborted; eRFID[67].bBottleTransferedToExit; eRFID[67].bBottleTransferedToLabeler; eRFID[67].lrWeightDif; eRFID[67].lrMinWeightCV;eRFID[67].lrMaxWeightCV;
eRFID[68].nCardNumber;eRFID[68].bROPPPuttedChecked;	eRFID[68].bROPPPutted;		eRFID[68].bROPPCapped;		eRFID[68].bROPPCappingAborted;eRFID[68].bROPPCappingOK; eRFID[68].bROPPCappingChecked;eRFID[68].bFormPresent; eRFID[68].bBottlePresent; eRFID[68].bDosingTwoPhases; eRFID[68].nDispencerNr; eRFID[68].nDispencerNrSecondPhase; eRFID[68].lrDoseVolumeSV; eRFID[68].lrDoseVolumeCV; eRFID[68].lrDoseVolumeSVSecondPhase; eRFID[68].lrDoseVolumeCVSecondPhase; eRFID[68].bDosed;	eRFID[68].bDoseAborted; eRFID[68].bWeighed; eRFID[68].lrWeightSV; eRFID[68].lrWeightCV; eRFID[68].lrWeightMeasuredCV; eRFID[68].bWeightOK; eRFID[68].bCapPutted; eRFID[68].bCapChecked; eRFID[68].bCapOK; eRFID[68].bCapGripperScrewed; eRFID[68].bCapGripperScrewAborted; eRFID[68].bBottleTransferedToExit; eRFID[68].bBottleTransferedToLabeler; eRFID[68].lrWeightDif; eRFID[68].lrMinWeightCV;eRFID[68].lrMaxWeightCV;
eRFID[69].nCardNumber;eRFID[69].bROPPPuttedChecked;	eRFID[69].bROPPPutted;		eRFID[69].bROPPCapped;		eRFID[69].bROPPCappingAborted;eRFID[69].bROPPCappingOK; eRFID[69].bROPPCappingChecked;eRFID[69].bFormPresent; eRFID[69].bBottlePresent; eRFID[69].bDosingTwoPhases; eRFID[69].nDispencerNr; eRFID[69].nDispencerNrSecondPhase; eRFID[69].lrDoseVolumeSV; eRFID[69].lrDoseVolumeCV; eRFID[69].lrDoseVolumeSVSecondPhase; eRFID[69].lrDoseVolumeCVSecondPhase; eRFID[69].bDosed;	eRFID[69].bDoseAborted; eRFID[69].bWeighed; eRFID[69].lrWeightSV; eRFID[69].lrWeightCV; eRFID[69].lrWeightMeasuredCV; eRFID[69].bWeightOK; eRFID[69].bCapPutted; eRFID[69].bCapChecked; eRFID[69].bCapOK; eRFID[69].bCapGripperScrewed; eRFID[69].bCapGripperScrewAborted; eRFID[69].bBottleTransferedToExit; eRFID[69].bBottleTransferedToLabeler; eRFID[69].lrWeightDif; eRFID[69].lrMinWeightCV;eRFID[69].lrMaxWeightCV;
eRFID[70].nCardNumber;eRFID[70].bROPPPuttedChecked;	eRFID[70].bROPPPutted;		eRFID[70].bROPPCapped;		eRFID[70].bROPPCappingAborted;eRFID[70].bROPPCappingOK; eRFID[70].bROPPCappingChecked;eRFID[70].bFormPresent; eRFID[70].bBottlePresent; eRFID[70].bDosingTwoPhases; eRFID[70].nDispencerNr; eRFID[70].nDispencerNrSecondPhase; eRFID[70].lrDoseVolumeSV; eRFID[70].lrDoseVolumeCV; eRFID[70].lrDoseVolumeSVSecondPhase; eRFID[70].lrDoseVolumeCVSecondPhase; eRFID[70].bDosed;	eRFID[70].bDoseAborted; eRFID[70].bWeighed; eRFID[70].lrWeightSV; eRFID[70].lrWeightCV; eRFID[70].lrWeightMeasuredCV; eRFID[70].bWeightOK; eRFID[70].bCapPutted; eRFID[70].bCapChecked; eRFID[70].bCapOK; eRFID[70].bCapGripperScrewed; eRFID[70].bCapGripperScrewAborted; eRFID[70].bBottleTransferedToExit; eRFID[70].bBottleTransferedToLabeler; eRFID[70].lrWeightDif; eRFID[70].lrMinWeightCV;eRFID[70].lrMaxWeightCV;
